QRS_NEXT_CUT()
PTP {E1 28616.934,E2 28616.934}
PTP {X 0,Y 607.906,A -85,B 0,C 180,E1 28616.934,E2 28616.934,E3 0,E4 0,E5 0,E6 0}
QRS_SPEED_INIT()
LIN {X 0,Y 607.906,Z 931,A -85,B 0,C 180,E1 28616.934,E2 28616.934,E3 0,E4 0,E5 0,E6 0} C_VEL
LIN {X 0,Y 607.906,Z 437.153,A -85,B 0,C 180,E1 28616.934,E2 28616.934} C_VEL
LIN {X 0,Y 607.906,Z 429.074,A -85,B 0,C 180,E1 28616.934,E2 28616.934} C_VEL
LIN {X 0,Y 607.894,Z 427.074,A -85,B 0,C 180,E1 28616.745,E2 28616.745} C_VEL
LIN {X 0,Y 607.905,Z 427.069,A -85,B 0,C 180,E1 28613.578,E2 28613.578} C_VEL
LIN {X 0,Y 607.887,Z 427.072,A -85,B 0,C 180,E1 28610.437,E2 28610.437} C_VEL
LIN {X 0,Y 607.904,Z 427.071,A -85,B 0,C 180,E1 28607.364,E2 28607.364} C_VEL
LIN {X 0,Y 607.887,Z 427.071,A -85,B 0,C 180,E1 28604.199,E2 28604.199} C_VEL
LIN {X 0,Y 607.905,Z 427.073,A -85,B 0,C 180,E1 28601.038,E2 28601.038} C_VEL
LIN {X 0,Y 607.891,Z 427.069,A -85,B 0,C 180,E1 28597.873,E2 28597.873} C_VEL
LIN {X 0,Y 607.916,Z 427.076,A -85,B 0,C 180,E1 28594.682,E2 28594.682} C_VEL
LIN {X 0,Y 607.915,Z 427.066,A -85,B 0,C 180,E1 28591.405,E2 28591.405} C_VEL
LIN {X 0,Y 607.89,Z 427.074,A -85,B 0,C 180,E1 28588.13,E2 28588.13} C_VEL
LIN {X 0,Y 607.908,Z 427.069,A -85,B 0,C 180,E1 28584.993,E2 28584.993} C_VEL
LIN {X 0,Y 607.885,Z 427.073,A -85,B 0,C 180,E1 28581.834,E2 28581.834} C_VEL
LIN {X 0,Y 607.906,Z 427.072,A -85,B 0,C 180,E1 28578.734,E2 28578.734} C_VEL
LIN {X 0,Y 607.913,Z 427.228,A -85,B 0,C 180,E1 28576.359,E2 28576.359} C_VEL
LIN {X 0,Y 607.865,Z 452.581,A -85,B 0,C 180,E1 28573.635,E2 28573.635} C_VEL
LIN {X 0,Y 607.881,Z 483.645,A -85,B 0,C 180,E1 28570.395,E2 28570.395} C_VEL
LIN {X 0,Y 607.891,Z 513.28,A -85,B 0,C 180,E1 28567.368,E2 28567.368} C_VEL
LIN {X 0,Y 607.869,Z 545.119,A -85,B 0,C 180,E1 28564.171,E2 28564.171} C_VEL
LIN {X 0,Y 607.907,Z 557.135,A -85,B 0,C 180,E1 28563.013,E2 28563.013} C_VEL
LIN {X 0,Y 607.887,Z 667.971,A -85,B 0,C 180,E1 28561.672,E2 28561.672} C_VEL
LIN {X 0,Y 607.914,Z 683.089,A -85,B 0,C 180,E1 28561.314,E2 28561.314} C_VEL
LIN {X 0,Y 607.919,Z 697.917,A -85,B 0,C 180,E1 28560.764,E2 28560.764} C_VEL
LIN {X 0,Y 607.887,Z 710.969,A -85,B 0,C 180,E1 28560.097,E2 28560.097} C_VEL
LIN {X 0,Y 607.919,Z 723.773,A -85,B 0,C 180,E1 28559.241,E2 28559.241} C_VEL
LIN {X 0,Y 607.918,Z 735.573,A -85,B 0,C 180,E1 28558.22,E2 28558.22} C_VEL
LIN {X 0,Y 607.918,Z 745.62,A -85,B 0,C 180,E1 28557.103,E2 28557.103} C_VEL
LIN {X 0,Y 607.916,Z 753.763,A -85,B 0,C 180,E1 28555.944,E2 28555.944} C_VEL
LIN {X 0,Y 607.918,Z 760.511,A -85,B 0,C 180,E1 28554.693,E2 28554.693} C_VEL
LIN {X 0,Y 607.918,Z 765.691,A -85,B 0,C 180,E1 28553.352,E2 28553.352} C_VEL
LIN {X 0,Y 607.917,Z 769.064,A -85,B 0,C 180,E1 28552.024,E2 28552.024} C_VEL
LIN {X 0,Y 607.917,Z 770.86,A -85,B 0,C 180,E1 28550.507,E2 28550.507} C_VEL
LIN {X 0,Y 607.916,Z 770.652,A -85,B 0,C 180,E1 28549.105,E2 28549.105} C_VEL
LIN {X 0,Y 607.915,Z 768.709,A -85,B 0,C 180,E1 28547.714,E2 28547.714} C_VEL
LIN {X 0,Y 607.919,Z 764.978,A -85,B 0,C 180,E1 28546.335,E2 28546.335} C_VEL
LIN {X 0,Y 607.919,Z 759.759,A -85,B 0,C 180,E1 28545.062,E2 28545.062} C_VEL
LIN {X 0,Y 607.918,Z 752.726,A -85,B 0,C 180,E1 28543.797,E2 28543.797} C_VEL
LIN {X 0,Y 607.919,Z 743.434,A -85,B 0,C 180,E1 28542.539,E2 28542.539} C_VEL
LIN {X 0,Y 607.917,Z 733.34,A -85,B 0,C 180,E1 28541.479,E2 28541.479} C_VEL
LIN {X 0,Y 607.917,Z 722.393,A -85,B 0,C 180,E1 28540.567,E2 28540.567} C_VEL
LIN {X 0,Y 607.901,Z 709.969,A -85,B 0,C 180,E1 28539.753,E2 28539.753} C_VEL
LIN {X 0,Y 607.919,Z 696.486,A -85,B 0,C 180,E1 28539.084,E2 28539.084} C_VEL
LIN {X 0,Y 607.919,Z 682.685,A -85,B 0,C 180,E1 28538.584,E2 28538.584} C_VEL
LIN {X 0,Y 607.915,Z 667.346,A -85,B 0,C 180,E1 28538.227,E2 28538.227} C_VEL
LIN {X 0,Y 607.917,Z 556.808,A -85,B 0,C 180,E1 28536.884,E2 28536.884} C_VEL
LIN {X 0,Y 607.915,Z 525.458,A -85,B 0,C 180,E1 28533.772,E2 28533.772} C_VEL
LIN {X 0,Y 607.88,Z 494.79,A -85,B 0,C 180,E1 28530.66,E2 28530.66} C_VEL
LIN {X 0,Y 607.901,Z 464.7,A -85,B 0,C 180,E1 28527.549,E2 28527.549} C_VEL
LIN {X 0,Y 607.919,Z 435.21,A -85,B 0,C 180,E1 28524.431,E2 28524.431} C_VEL
LIN {X 0,Y 607.9,Z 427.179,A -85,B 0,C 180,E1 28523.531,E2 28523.531} C_VEL
LIN {X 0,Y 607.841,Z 427.076,A -85,B 0,C 180,E1 28520.628,E2 28520.628} C_VEL
LIN {X 0,Y 607.911,Z 427.078,A -85,B 0,C 180,E1 28517.557,E2 28517.557} C_VEL
LIN {X 0,Y 607.836,Z 427.076,A -85,B 0,C 180,E1 28514.545,E2 28514.545} C_VEL
LIN {X 0,Y 607.919,Z 427.077,A -85,B 0,C 180,E1 28511.492,E2 28511.492} C_VEL
LIN {X 0,Y 607.831,Z 427.077,A -85,B 0,C 180,E1 28508.48,E2 28508.48} C_VEL
LIN {X 0,Y 607.906,Z 427.077,A -85,B 0,C 180,E1 28505.444,E2 28505.444} C_VEL
LIN {X 0,Y 607.827,Z 427.077,A -85,B 0,C 180,E1 28502.455,E2 28502.455} C_VEL
LIN {X 0,Y 607.883,Z 427.077,A -85,B 0,C 180,E1 28499.53,E2 28499.53} C_VEL
LIN {X 0,Y 607.829,Z 427.077,A -85,B 0,C 180,E1 28496.447,E2 28496.447} C_VEL
LIN {X 0,Y 607.87,Z 427.077,A -85,B 0,C 180,E1 28493.547,E2 28493.547} C_VEL
LIN {X 0,Y 607.839,Z 427.077,A -85,B 0,C 180,E1 28490.462,E2 28490.462} C_VEL
LIN {X 0,Y 607.846,Z 427.077,A -85,B 0,C 180,E1 28487.718,E2 28487.718} C_VEL
LIN {X 0,Y 607.85,Z 427.076,A -85,B 0,C 180,E1 28484.447,E2 28484.447} C_VEL
LIN {X 0,Y 607.848,Z 427.076,A -85,B 0,C 180,E1 28481.648,E2 28481.648} C_VEL
LIN {X 0,Y 607.853,Z 427.075,A -85,B 0,C 180,E1 28478.314,E2 28478.314} C_VEL
LIN {X 0,Y 607.856,Z 427.076,A -85,B 0,C 180,E1 28475.489,E2 28475.489} C_VEL
LIN {X 0,Y 607.857,Z 427.074,A -85,B 0,C 180,E1 28472.205,E2 28472.205} C_VEL
LIN {X 0,Y 607.864,Z 427.076,A -85,B 0,C 180,E1 28469.333,E2 28469.333} C_VEL
LIN {X 0,Y 607.859,Z 427.073,A -85,B 0,C 180,E1 28466.052,E2 28466.052} C_VEL
LIN {X 0,Y 607.875,Z 427.076,A -85,B 0,C 180,E1 28463.149,E2 28463.149} C_VEL
LIN {X 0,Y 607.86,Z 427.073,A -85,B 0,C 180,E1 28459.907,E2 28459.907} C_VEL
LIN {X 0,Y 607.891,Z 427.076,A -85,B 0,C 180,E1 28456.926,E2 28456.926} C_VEL
LIN {X 0,Y 607.86,Z 427.073,A -85,B 0,C 180,E1 28453.702,E2 28453.702} C_VEL
LIN {X 0,Y 607.908,Z 427.077,A -85,B 0,C 180,E1 28450.711,E2 28450.711} C_VEL
LIN {X 0,Y 607.863,Z 427.072,A -85,B 0,C 180,E1 28447.562,E2 28447.562} C_VEL
LIN {X 0,Y 607.911,Z 427.078,A -85,B 0,C 180,E1 28444.528,E2 28444.528} C_VEL
LIN {X 0,Y 607.866,Z 427.072,A -85,B 0,C 180,E1 28441.414,E2 28441.414} C_VEL
LIN {X 0,Y 607.915,Z 427.075,A -85,B 0,C 180,E1 28438.304,E2 28438.304} C_VEL
LIN {X 0,Y 607.867,Z 427.073,A -85,B 0,C 180,E1 28435.188,E2 28435.188} C_VEL
LIN {X 0,Y 607.913,Z 427.072,A -85,B 0,C 180,E1 28432.059,E2 28432.059} C_VEL
LIN {X 0,Y 607.87,Z 427.073,A -85,B 0,C 180,E1 28429,E2 28429} C_VEL
LIN {X 0,Y 607.912,Z 427.071,A -85,B 0,C 180,E1 28425.912,E2 28425.912} C_VEL
LIN {X 0,Y 607.875,Z 427.073,A -85,B 0,C 180,E1 28422.874,E2 28422.874} C_VEL
LIN {X 0,Y 607.912,Z 427.069,A -85,B 0,C 180,E1 28419.694,E2 28419.694} C_VEL
LIN {X 0,Y 607.885,Z 427.074,A -85,B 0,C 180,E1 28416.544,E2 28416.544} C_VEL
LIN {X 0,Y 607.904,Z 427.067,A -85,B 0,C 180,E1 28413.267,E2 28413.267} C_VEL
LIN {X 0,Y 607.915,Z 427.076,A -85,B 0,C 180,E1 28410,E2 28410} C_VEL
LIN {X 0,Y 607.885,Z 427.07,A -85,B 0,C 180,E1 28406.789,E2 28406.789} C_VEL
LIN {X 0,Y 607.906,Z 427.073,A -85,B 0,C 180,E1 28403.693,E2 28403.693} C_VEL
LIN {X 0,Y 607.886,Z 427.071,A -85,B 0,C 180,E1 28400.588,E2 28400.588} C_VEL
LIN {X 0,Y 607.903,Z 427.072,A -85,B 0,C 180,E1 28397.465,E2 28397.465} C_VEL
LIN {X 0,Y 607.889,Z 427.073,A -85,B 0,C 180,E1 28394.317,E2 28394.317} C_VEL
LIN {X 0,Y 607.906,Z 427.069,A -85,B 0,C 180,E1 28391.123,E2 28391.123} C_VEL
LIN {X 0,Y 607.902,Z 427.075,A -85,B 0,C 180,E1 28387.963,E2 28387.963} C_VEL
LIN {X 0,Y 607.909,Z 427.067,A -85,B 0,C 180,E1 28384.677,E2 28384.677} C_VEL
LIN {X 0,Y 607.902,Z 427.076,A -85,B 0,C 180,E1 28381.426,E2 28381.426} C_VEL
LIN {X 0,Y 607.906,Z 427.311,A -85,B 0,C 180,E1 28379.783,E2 28379.783} C_VEL
LIN {X 0,Y 607.918,Z 435.341,A -85,B 0,C 180,E1 28379.195,E2 28379.195} C_VEL
LIN {X 0,Y 607.898,Z 480.356,A -85,B 0,C 180,E1 28376.155,E2 28376.155} C_VEL
LIN {X 0,Y 607.881,Z 526.04,A -85,B 0,C 180,E1 28373.149,E2 28373.149} C_VEL
LIN {X 0,Y 607.914,Z 539.004,A -85,B 0,C 180,E1 28372.33,E2 28372.33} C_VEL
LIN {X 0,Y 607.912,Z 748.311,A -85,B 0,C 180,E1 28369.705,E2 28369.705} C_VEL
LIN {X 0,Y 607.888,Z 766.586,A -85,B 0,C 180,E1 28369.306,E2 28369.306} C_VEL
LIN {X 0,Y 607.901,Z 784.762,A -85,B 0,C 180,E1 28368.732,E2 28368.732} C_VEL
LIN {X 0,Y 607.893,Z 803.057,A -85,B 0,C 180,E1 28367.963,E2 28367.963} C_VEL
LIN {X 0,Y 607.919,Z 819.788,A -85,B 0,C 180,E1 28367.073,E2 28367.073} C_VEL
LIN {X 0,Y 607.916,Z 835.64,A -85,B 0,C 180,E1 28366.041,E2 28366.041} C_VEL
LIN {X 0,Y 607.917,Z 850.561,A -85,B 0,C 180,E1 28364.867,E2 28364.867} C_VEL
LIN {X 0,Y 607.918,Z 864.218,A -85,B 0,C 180,E1 28363.582,E2 28363.582} C_VEL
LIN {X 0,Y 607.918,Z 876.905,A -85,B 0,C 180,E1 28362.153,E2 28362.153} C_VEL
LIN {X 0,Y 607.911,Z 888.224,A -85,B 0,C 180,E1 28360.615,E2 28360.615} C_VEL
LIN {X 0,Y 607.918,Z 897.988,A -85,B 0,C 180,E1 28358.989,E2 28358.989} C_VEL
LIN {X 0,Y 607.909,Z 905.863,A -85,B 0,C 180,E1 28357.35,E2 28357.35} C_VEL
LIN {X 0,Y 607.906,Z 912.107,A -85,B 0,C 180,E1 28355.664,E2 28355.664} C_VEL
LIN {X 0,Y 607.917,Z 916.872,A -85,B 0,C 180,E1 28353.867,E2 28353.867} C_VEL
LIN {X 0,Y 607.916,Z 919.787,A -85,B 0,C 180,E1 28352.074,E2 28352.074} C_VEL
LIN {X 0,Y 607.907,Z 920.94,A -85,B 0,C 180,E1 28350.283,E2 28350.283} C_VEL
LIN {X 0,Y 607.915,Z 920.348,A -85,B 0,C 180,E1 28348.492,E2 28348.492} C_VEL
LIN {X 0,Y 607.908,Z 918.005,A -85,B 0,C 180,E1 28346.7,E2 28346.7} C_VEL
LIN {X 0,Y 607.905,Z 914.096,A -85,B 0,C 180,E1 28344.999,E2 28344.999} C_VEL
LIN {X 0,Y 607.912,Z 908.468,A -85,B 0,C 180,E1 28343.294,E2 28343.294} C_VEL
LIN {X 0,Y 607.915,Z 901.423,A -85,B 0,C 180,E1 28341.678,E2 28341.678} C_VEL
LIN {X 0,Y 607.911,Z 892.509,A -85,B 0,C 180,E1 28340.055,E2 28340.055} C_VEL
LIN {X 0,Y 607.919,Z 882.145,A -85,B 0,C 180,E1 28338.521,E2 28338.521} C_VEL
LIN {X 0,Y 607.914,Z 870.346,A -85,B 0,C 180,E1 28337.075,E2 28337.075} C_VEL
LIN {X 0,Y 607.917,Z 857.089,A -85,B 0,C 180,E1 28335.717,E2 28335.717} C_VEL
LIN {X 0,Y 607.917,Z 842.235,A -85,B 0,C 180,E1 28334.449,E2 28334.449} C_VEL
LIN {X 0,Y 607.917,Z 826.219,A -85,B 0,C 180,E1 28333.321,E2 28333.321} C_VEL
LIN {X 0,Y 607.898,Z 810.027,A -85,B 0,C 180,E1 28332.384,E2 28332.384} C_VEL
LIN {X 0,Y 607.913,Z 793.065,A -85,B 0,C 180,E1 28331.592,E2 28331.592} C_VEL
LIN {X 0,Y 607.886,Z 775.227,A -85,B 0,C 180,E1 28330.944,E2 28330.944} C_VEL
LIN {X 0,Y 607.899,Z 756.387,A -85,B 0,C 180,E1 28330.45,E2 28330.45} C_VEL
LIN {X 0,Y 607.919,Z 736.792,A -85,B 0,C 180,E1 28330.128,E2 28330.128} C_VEL
LIN {X 0,Y 607.915,Z 538.331,A -85,B 0,C 180,E1 28327.645,E2 28327.645} C_VEL
LIN {X 0,Y 607.904,Z 491.389,A -85,B 0,C 180,E1 28324.578,E2 28324.578} C_VEL
LIN {X 0,Y 607.919,Z 444.131,A -85,B 0,C 180,E1 28321.405,E2 28321.405} C_VEL
LIN {X 0,Y 607.907,Z 427.395,A -85,B 0,C 180,E1 28320.232,E2 28320.232} C_VEL
LIN {X 0,Y 607.912,Z 427.067,A -85,B 0,C 180,E1 28319.339,E2 28319.339} C_VEL
LIN {X 0,Y 607.906,Z 427.076,A -85,B 0,C 180,E1 28316.112,E2 28316.112} C_VEL
LIN {X 0,Y 607.902,Z 427.069,A -85,B 0,C 180,E1 28312.912,E2 28312.912} C_VEL
LIN {X 0,Y 607.895,Z 427.073,A -85,B 0,C 180,E1 28309.729,E2 28309.729} C_VEL
LIN {X 0,Y 607.898,Z 427.071,A -85,B 0,C 180,E1 28306.566,E2 28306.566} C_VEL
LIN {X 0,Y 607.893,Z 427.071,A -85,B 0,C 180,E1 28303.434,E2 28303.434} C_VEL
LIN {X 0,Y 607.901,Z 427.073,A -85,B 0,C 180,E1 28300.27,E2 28300.27} C_VEL
LIN {X 0,Y 607.899,Z 427.068,A -85,B 0,C 180,E1 28297.088,E2 28297.088} C_VEL
LIN {X 0,Y 607.913,Z 427.078,A -85,B 0,C 180,E1 28293.84,E2 28293.84} C_VEL
LIN {X 0,Y 607.908,Z 427.067,A -85,B 0,C 180,E1 28290.546,E2 28290.546} C_VEL
LIN {X 0,Y 607.894,Z 427.073,A -85,B 0,C 180,E1 28287.316,E2 28287.316} C_VEL
LIN {X 0,Y 607.901,Z 427.07,A -85,B 0,C 180,E1 28284.176,E2 28284.176} C_VEL
LIN {X 0,Y 607.891,Z 427.071,A -85,B 0,C 180,E1 28281.012,E2 28281.012} C_VEL
LIN {X 0,Y 607.901,Z 427.072,A -85,B 0,C 180,E1 28277.913,E2 28277.913} C_VEL
LIN {X 0,Y 607.89,Z 427.071,A -85,B 0,C 180,E1 28274.868,E2 28274.868} C_VEL
LIN {X 0,Y 607.9,Z 427.072,A -85,B 0,C 180,E1 28271.768,E2 28271.768} C_VEL
LIN {X 0,Y 607.89,Z 427.071,A -85,B 0,C 180,E1 28268.688,E2 28268.688} C_VEL
LIN {X 0,Y 607.903,Z 427.073,A -85,B 0,C 180,E1 28265.569,E2 28265.569} C_VEL
LIN {X 0,Y 607.892,Z 427.07,A -85,B 0,C 180,E1 28262.451,E2 28262.451} C_VEL
LIN {X 0,Y 607.91,Z 427.076,A -85,B 0,C 180,E1 28259.246,E2 28259.246} C_VEL
LIN {X 0,Y 607.894,Z 427.074,A -85,B 0,C 180,E1 28256.745,E2 28256.745} C_VEL
LIN {X 0,Y 606.888,Z 427.198,A -85,B 0,C 180,E1 28256.019,E2 28256.019} C_VEL
LIN {X 0,Y 600.49,Z 427.993,A -85,B 0,C 180,E1 28253.983,E2 28253.983} C_VEL
LIN {X 0,Y 599.964,Z 428.06,A -85,B 0,C 180,E1 28253.453,E2 28253.453} C_VEL
LIN {X 0,Y 599.949,Z 428.059,A -85,B 0,C 180,E1 28250.309,E2 28250.309} C_VEL
LIN {X 0,Y 599.968,Z 428.063,A -85,B 0,C 180,E1 28247.096,E2 28247.096} C_VEL
LIN {X 0,Y 599.962,Z 428.057,A -85,B 0,C 180,E1 28243.84,E2 28243.84} C_VEL
LIN {X 0,Y 599.961,Z 428.064,A -85,B 0,C 180,E1 28240.53,E2 28240.53} C_VEL
LIN {X 0,Y 599.973,Z 428.057,A -85,B 0,C 180,E1 28237.358,E2 28237.358} C_VEL
LIN {X 0,Y 599.948,Z 428.062,A -85,B 0,C 180,E1 28234.151,E2 28234.151} C_VEL
LIN {X 0,Y 599.966,Z 428.06,A -85,B 0,C 180,E1 28230.99,E2 28230.99} C_VEL
LIN {X 0,Y 599.946,Z 428.06,A -85,B 0,C 180,E1 28227.846,E2 28227.846} C_VEL
LIN {X 0,Y 599.969,Z 428.063,A -85,B 0,C 180,E1 28224.67,E2 28224.67} C_VEL
LIN {X 0,Y 599.949,Z 428.06,A -85,B 0,C 180,E1 28221.563,E2 28221.563} C_VEL
LIN {X 0,Y 599.977,Z 428.065,A -85,B 0,C 180,E1 28218.296,E2 28218.296} C_VEL
LIN {X 0,Y 600.001,Z 428.308,A -85,B 0,C 180,E1 28216.611,E2 28216.611} C_VEL
LIN {X 0,Y 600.305,Z 432.323,A -85,B 0,C 180,E1 28216.141,E2 28216.141} C_VEL
LIN {X 0,Y 600.213,Z 462.032,A -85,B 0,C 180,E1 28212.947,E2 28212.947} C_VEL
LIN {X 0,Y 600.131,Z 492.243,A -85,B 0,C 180,E1 28209.774,E2 28209.774} C_VEL
LIN {X 0,Y 600.074,Z 523.353,A -85,B 0,C 180,E1 28206.57,E2 28206.57} C_VEL
LIN {X 0,Y 599.98,Z 553.885,A -85,B 0,C 180,E1 28203.477,E2 28203.477} C_VEL
LIN {X 0,Y 600.063,Z 557.379,A -85,B 0,C 180,E1 28203.181,E2 28203.181} C_VEL
LIN {X 0,Y 600.05,Z 668.429,A -85,B 0,C 180,E1 28201.819,E2 28201.819} C_VEL
LIN {X 0,Y 600.059,Z 683.234,A -85,B 0,C 180,E1 28201.461,E2 28201.461} C_VEL
LIN {X 0,Y 600.039,Z 698.352,A -85,B 0,C 180,E1 28200.889,E2 28200.889} C_VEL
LIN {X 0,Y 599.979,Z 711.224,A -85,B 0,C 180,E1 28200.217,E2 28200.217} C_VEL
LIN {X 0,Y 599.985,Z 723.853,A -85,B 0,C 180,E1 28199.358,E2 28199.358} C_VEL
LIN {X 0,Y 599.959,Z 735.895,A -85,B 0,C 180,E1 28198.298,E2 28198.298} C_VEL
LIN {X 0,Y 599.941,Z 746.161,A -85,B 0,C 180,E1 28197.131,E2 28197.131} C_VEL
LIN {X 0,Y 599.927,Z 754.564,A -85,B 0,C 180,E1 28195.891,E2 28195.891} C_VEL
LIN {X 0,Y 599.921,Z 761.097,A -85,B 0,C 180,E1 28194.624,E2 28194.624} C_VEL
LIN {X 0,Y 599.915,Z 766.428,A -85,B 0,C 180,E1 28193.162,E2 28193.162} C_VEL
LIN {X 0,Y 599.916,Z 769.618,A -85,B 0,C 180,E1 28191.715,E2 28191.715} C_VEL
LIN {X 0,Y 599.919,Z 770.906,A -85,B 0,C 180,E1 28190.385,E2 28190.385} C_VEL
LIN {X 0,Y 599.914,Z 770.563,A -85,B 0,C 180,E1 28188.965,E2 28188.965} C_VEL
LIN {X 0,Y 599.915,Z 768.439,A -85,B 0,C 180,E1 28187.558,E2 28187.558} C_VEL
LIN {X 0,Y 599.919,Z 764.544,A -85,B 0,C 180,E1 28186.16,E2 28186.16} C_VEL
LIN {X 0,Y 599.921,Z 758.689,A -85,B 0,C 180,E1 28184.773,E2 28184.773} C_VEL
LIN {X 0,Y 599.932,Z 751.258,A -85,B 0,C 180,E1 28183.493,E2 28183.493} C_VEL
LIN {X 0,Y 599.948,Z 742.392,A -85,B 0,C 180,E1 28182.317,E2 28182.317} C_VEL
LIN {X 0,Y 599.969,Z 731.526,A -85,B 0,C 180,E1 28181.195,E2 28181.195} C_VEL
LIN {X 0,Y 599.992,Z 719.4,A -85,B 0,C 180,E1 28180.223,E2 28180.223} C_VEL
LIN {X 0,Y 600.009,Z 706.382,A -85,B 0,C 180,E1 28179.419,E2 28179.419} C_VEL
LIN {X 0,Y 600.047,Z 693.632,A -85,B 0,C 180,E1 28178.818,E2 28178.818} C_VEL
LIN {X 0,Y 600.068,Z 678.136,A -85,B 0,C 180,E1 28178.305,E2 28178.305} C_VEL
LIN {X 0,Y 600.083,Z 663.073,A -85,B 0,C 180,E1 28178.006,E2 28178.006} C_VEL
LIN {X 0,Y 600.032,Z 556.838,A -85,B 0,C 180,E1 28176.712,E2 28176.712} C_VEL
LIN {X 0,Y 600.07,Z 525.261,A -85,B 0,C 180,E1 28173.534,E2 28173.534} C_VEL
LIN {X 0,Y 600.129,Z 493.692,A -85,B 0,C 180,E1 28170.286,E2 28170.286} C_VEL
LIN {X 0,Y 600.201,Z 463.661,A -85,B 0,C 180,E1 28167.135,E2 28167.135} C_VEL
LIN {X 0,Y 600.301,Z 434.227,A -85,B 0,C 180,E1 28163.977,E2 28163.977} C_VEL
LIN {X 0,Y 600.118,Z 429.008,A -85,B 0,C 180,E1 28163.398,E2 28163.398} C_VEL
LIN {X 0,Y 599.928,Z 428.099,A -85,B 0,C 180,E1 28163.204,E2 28163.204} C_VEL
LIN {X 0,Y 599.916,Z 428.065,A -85,B 0,C 180,E1 28160.309,E2 28160.309} C_VEL
LIN {X 0,Y 599.912,Z 428.066,A -85,B 0,C 180,E1 28156.997,E2 28156.997} C_VEL
LIN {X 0,Y 599.916,Z 428.065,A -85,B 0,C 180,E1 28154.137,E2 28154.137} C_VEL
LIN {X 0,Y 599.903,Z 428.066,A -85,B 0,C 180,E1 28150.832,E2 28150.832} C_VEL
LIN {X 0,Y 599.907,Z 428.065,A -85,B 0,C 180,E1 28148.078,E2 28148.078} C_VEL
LIN {X 0,Y 599.901,Z 428.066,A -85,B 0,C 180,E1 28144.743,E2 28144.743} C_VEL
LIN {X 0,Y 599.903,Z 428.066,A -85,B 0,C 180,E1 28141.965,E2 28141.965} C_VEL
LIN {X 0,Y 599.898,Z 428.066,A -85,B 0,C 180,E1 28138.667,E2 28138.667} C_VEL
LIN {X 0,Y 599.897,Z 428.066,A -85,B 0,C 180,E1 28135.931,E2 28135.931} C_VEL
LIN {X 0,Y 599.909,Z 428.065,A -85,B 0,C 180,E1 28132.65,E2 28132.65} C_VEL
LIN {X 0,Y 599.901,Z 428.066,A -85,B 0,C 180,E1 28129.833,E2 28129.833} C_VEL
LIN {X 0,Y 599.92,Z 428.065,A -85,B 0,C 180,E1 28126.608,E2 28126.608} C_VEL
LIN {X 0,Y 599.904,Z 428.065,A -85,B 0,C 180,E1 28123.764,E2 28123.764} C_VEL
LIN {X 0,Y 599.929,Z 428.063,A -85,B 0,C 180,E1 28120.537,E2 28120.537} C_VEL
LIN {X 0,Y 599.908,Z 428.065,A -85,B 0,C 180,E1 28117.657,E2 28117.657} C_VEL
LIN {X 0,Y 599.931,Z 428.061,A -85,B 0,C 180,E1 28114.402,E2 28114.402} C_VEL
LIN {X 0,Y 599.911,Z 428.065,A -85,B 0,C 180,E1 28111.557,E2 28111.557} C_VEL
LIN {X 0,Y 599.942,Z 428.061,A -85,B 0,C 180,E1 28108.358,E2 28108.358} C_VEL
LIN {X 0,Y 599.918,Z 428.063,A -85,B 0,C 180,E1 28105.4,E2 28105.4} C_VEL
LIN {X 0,Y 599.93,Z 428.062,A -85,B 0,C 180,E1 28102.082,E2 28102.082} C_VEL
LIN {X 0,Y 599.937,Z 428.064,A -85,B 0,C 180,E1 28099.096,E2 28099.096} C_VEL
LIN {X 0,Y 599.926,Z 428.061,A -85,B 0,C 180,E1 28095.863,E2 28095.863} C_VEL
LIN {X 0,Y 599.96,Z 428.066,A -85,B 0,C 180,E1 28092.806,E2 28092.806} C_VEL
LIN {X 0,Y 599.924,Z 428.06,A -85,B 0,C 180,E1 28089.594,E2 28089.594} C_VEL
LIN {X 0,Y 599.976,Z 428.065,A -85,B 0,C 180,E1 28086.507,E2 28086.507} C_VEL
LIN {X 0,Y 599.925,Z 428.062,A -85,B 0,C 180,E1 28083.32,E2 28083.32} C_VEL
LIN {X 0,Y 599.975,Z 428.06,A -85,B 0,C 180,E1 28080.191,E2 28080.191} C_VEL
LIN {X 0,Y 599.928,Z 428.062,A -85,B 0,C 180,E1 28077.134,E2 28077.134} C_VEL
LIN {X 0,Y 599.977,Z 428.058,A -85,B 0,C 180,E1 28073.974,E2 28073.974} C_VEL
LIN {X 0,Y 599.934,Z 428.062,A -85,B 0,C 180,E1 28070.89,E2 28070.89} C_VEL
LIN {X 0,Y 599.975,Z 428.057,A -85,B 0,C 180,E1 28067.684,E2 28067.684} C_VEL
LIN {X 0,Y 599.961,Z 428.064,A -85,B 0,C 180,E1 28064.421,E2 28064.421} C_VEL
LIN {X 0,Y 599.942,Z 428.06,A -85,B 0,C 180,E1 28061.136,E2 28061.136} C_VEL
LIN {X 0,Y 599.972,Z 428.063,A -85,B 0,C 180,E1 28057.978,E2 28057.978} C_VEL
LIN {X 0,Y 599.941,Z 428.061,A -85,B 0,C 180,E1 28054.819,E2 28054.819} C_VEL
LIN {X 0,Y 599.97,Z 428.06,A -85,B 0,C 180,E1 28051.644,E2 28051.644} C_VEL
LIN {X 0,Y 599.945,Z 428.061,A -85,B 0,C 180,E1 28048.558,E2 28048.558} C_VEL
LIN {X 0,Y 599.971,Z 428.057,A -85,B 0,C 180,E1 28045.37,E2 28045.37} C_VEL
LIN {X 0,Y 599.96,Z 428.064,A -85,B 0,C 180,E1 28042.173,E2 28042.173} C_VEL
LIN {X 0,Y 599.959,Z 428.058,A -85,B 0,C 180,E1 28038.831,E2 28038.831} C_VEL
LIN {X 0,Y 599.968,Z 428.063,A -85,B 0,C 180,E1 28035.638,E2 28035.638} C_VEL
LIN {X 0,Y 599.951,Z 428.061,A -85,B 0,C 180,E1 28032.414,E2 28032.414} C_VEL
LIN {X 0,Y 599.962,Z 428.061,A -85,B 0,C 180,E1 28029.293,E2 28029.293} C_VEL
LIN {X 0,Y 599.954,Z 428.063,A -85,B 0,C 180,E1 28026.155,E2 28026.155} C_VEL
LIN {X 0,Y 599.968,Z 428.056,A -85,B 0,C 180,E1 28022.908,E2 28022.908} C_VEL
LIN {X 0,Y 599.982,Z 428.256,A -85,B 0,C 180,E1 28020.157,E2 28020.157} C_VEL
LIN {X 0,Y 600.653,Z 431.523,A -85,B 0,C 180,E1 28019.85,E2 28019.85} C_VEL
LIN {X 0,Y 600.505,Z 477.206,A -85,B 0,C 180,E1 28016.716,E2 28016.716} C_VEL
LIN {X 0,Y 600.351,Z 524.464,A -85,B 0,C 180,E1 28013.56,E2 28013.56} C_VEL
LIN {X 0,Y 600.433,Z 539.199,A -85,B 0,C 180,E1 28012.62,E2 28012.62} C_VEL
LIN {X 0,Y 600.372,Z 748.311,A -85,B 0,C 180,E1 28009.963,E2 28009.963} C_VEL
LIN {X 0,Y 600.309,Z 767.215,A -85,B 0,C 180,E1 28009.541,E2 28009.541} C_VEL
LIN {X 0,Y 600.273,Z 785.404,A -85,B 0,C 180,E1 28008.954,E2 28008.954} C_VEL
LIN {X 0,Y 600.211,Z 803.054,A -85,B 0,C 180,E1 28008.201,E2 28008.201} C_VEL
LIN {X 0,Y 600.18,Z 819.704,A -85,B 0,C 180,E1 28007.305,E2 28007.305} C_VEL
LIN {X 0,Y 600.122,Z 835.639,A -85,B 0,C 180,E1 28006.255,E2 28006.255} C_VEL
LIN {X 0,Y 600.069,Z 850.562,A -85,B 0,C 180,E1 28005.066,E2 28005.066} C_VEL
LIN {X 0,Y 600.02,Z 864.018,A -85,B 0,C 180,E1 28003.786,E2 28003.786} C_VEL
LIN {X 0,Y 599.985,Z 876.906,A -85,B 0,C 180,E1 28002.316,E2 28002.316} C_VEL
LIN {X 0,Y 599.953,Z 888.224,A -85,B 0,C 180,E1 28000.758,E2 28000.758} C_VEL
LIN {X 0,Y 599.935,Z 897.989,A -85,B 0,C 180,E1 27999.11,E2 27999.11} C_VEL
LIN {X 0,Y 599.92,Z 906.042,A -85,B 0,C 180,E1 27997.406,E2 27997.406} C_VEL
LIN {X 0,Y 599.91,Z 912.409,A -85,B 0,C 180,E1 27995.643,E2 27995.643} C_VEL
LIN {X 0,Y 599.918,Z 916.873,A -85,B 0,C 180,E1 27993.918,E2 27993.918} C_VEL
LIN {X 0,Y 599.917,Z 919.787,A -85,B 0,C 180,E1 27992.101,E2 27992.101} C_VEL
LIN {X 0,Y 599.907,Z 920.94,A -85,B 0,C 180,E1 27990.287,E2 27990.287} C_VEL
LIN {X 0,Y 599.915,Z 920.348,A -85,B 0,C 180,E1 27988.472,E2 27988.472} C_VEL
LIN {X 0,Y 599.907,Z 918.006,A -85,B 0,C 180,E1 27986.656,E2 27986.656} C_VEL
LIN {X 0,Y 599.908,Z 914.097,A -85,B 0,C 180,E1 27984.932,E2 27984.932} C_VEL
LIN {X 0,Y 599.919,Z 908.468,A -85,B 0,C 180,E1 27983.204,E2 27983.204} C_VEL
LIN {X 0,Y 599.927,Z 901.424,A -85,B 0,C 180,E1 27981.567,E2 27981.567} C_VEL
LIN {X 0,Y 599.942,Z 892.51,A -85,B 0,C 180,E1 27979.922,E2 27979.922} C_VEL
LIN {X 0,Y 599.969,Z 882.146,A -85,B 0,C 180,E1 27978.367,E2 27978.367} C_VEL
LIN {X 0,Y 600,Z 870.347,A -85,B 0,C 180,E1 27976.901,E2 27976.901} C_VEL
LIN {X 0,Y 600.049,Z 856.752,A -85,B 0,C 180,E1 27975.493,E2 27975.493} C_VEL
LIN {X 0,Y 600.103,Z 842.234,A -85,B 0,C 180,E1 27974.242,E2 27974.242} C_VEL
LIN {X 0,Y 600.164,Z 826.222,A -85,B 0,C 180,E1 27973.1,E2 27973.1} C_VEL
LIN {X 0,Y 600.199,Z 809.035,A -85,B 0,C 180,E1 27972.1,E2 27972.1} C_VEL
LIN {X 0,Y 600.279,Z 791.772,A -85,B 0,C 180,E1 27971.298,E2 27971.298} C_VEL
LIN {X 0,Y 600.297,Z 773.83,A -85,B 0,C 180,E1 27970.652,E2 27970.652} C_VEL
LIN {X 0,Y 600.353,Z 755.31,A -85,B 0,C 180,E1 27970.173,E2 27970.173} C_VEL
LIN {X 0,Y 600.395,Z 735.522,A -85,B 0,C 180,E1 27969.853,E2 27969.853} C_VEL
LIN {X 0,Y 600.381,Z 538.736,A -85,B 0,C 180,E1 27967.368,E2 27967.368} C_VEL
LIN {X 0,Y 600.472,Z 490.601,A -85,B 0,C 180,E1 27964.188,E2 27964.188} C_VEL
LIN {X 0,Y 600.612,Z 444.131,A -85,B 0,C 180,E1 27961.025,E2 27961.025} C_VEL
LIN {X 0,Y 600.43,Z 429.953,A -85,B 0,C 180,E1 27960.029,E2 27960.029} C_VEL
LIN {X 0,Y 599.968,Z 428.159,A -85,B 0,C 180,E1 27959.813,E2 27959.813} C_VEL
LIN {X 0,Y 599.96,Z 428.063,A -85,B 0,C 180,E1 27956.636,E2 27956.636} C_VEL
LIN {X 0,Y 599.963,Z 428.058,A -85,B 0,C 180,E1 27953.443,E2 27953.443} C_VEL
LIN {X 0,Y 599.974,Z 428.066,A -85,B 0,C 180,E1 27950.198,E2 27950.198} C_VEL
LIN {X 0,Y 599.969,Z 428.056,A -85,B 0,C 180,E1 27946.881,E2 27946.881} C_VEL
LIN {X 0,Y 599.958,Z 428.063,A -85,B 0,C 180,E1 27943.674,E2 27943.674} C_VEL
LIN {X 0,Y 599.961,Z 428.059,A -85,B 0,C 180,E1 27940.538,E2 27940.538} C_VEL
LIN {X 0,Y 599.955,Z 428.06,A -85,B 0,C 180,E1 27937.346,E2 27937.346} C_VEL
LIN {X 0,Y 599.963,Z 428.062,A -85,B 0,C 180,E1 27934.168,E2 27934.168} C_VEL
LIN {X 0,Y 599.958,Z 428.058,A -85,B 0,C 180,E1 27930.995,E2 27930.995} C_VEL
LIN {X 0,Y 599.973,Z 428.066,A -85,B 0,C 180,E1 27927.707,E2 27927.707} C_VEL
LIN {X 0,Y 599.971,Z 428.056,A -85,B 0,C 180,E1 27924.412,E2 27924.412} C_VEL
LIN {X 0,Y 599.955,Z 428.062,A -85,B 0,C 180,E1 27921.201,E2 27921.201} C_VEL
LIN {X 0,Y 599.963,Z 428.059,A -85,B 0,C 180,E1 27918.058,E2 27918.058} C_VEL
LIN {X 0,Y 599.952,Z 428.06,A -85,B 0,C 180,E1 27914.97,E2 27914.97} C_VEL
LIN {X 0,Y 599.962,Z 428.061,A -85,B 0,C 180,E1 27911.828,E2 27911.828} C_VEL
LIN {X 0,Y 599.951,Z 428.06,A -85,B 0,C 180,E1 27908.723,E2 27908.723} C_VEL
LIN {X 0,Y 599.965,Z 428.062,A -85,B 0,C 180,E1 27905.547,E2 27905.547} C_VEL
LIN {X 0,Y 599.955,Z 428.058,A -85,B 0,C 180,E1 27902.388,E2 27902.388} C_VEL
LIN {X 0,Y 599.973,Z 428.066,A -85,B 0,C 180,E1 27899.14,E2 27899.14} C_VEL
LIN {X 0,Y 599.971,Z 428.056,A -85,B 0,C 180,E1 27895.795,E2 27895.795} C_VEL
LIN {X 0,Y 599.964,Z 428.06,A -85,B 0,C 180,E1 27893.453,E2 27893.453} C_VEL
LIN {X 0,Y 598.972,Z 428.19,A -85,B 0,C 180,E1 27892.717,E2 27892.717} C_VEL
LIN {X 0,Y 592.53,Z 428.989,A -85,B 0,C 180,E1 27890.653,E2 27890.653} C_VEL
LIN {X 0,Y 592.015,Z 429.046,A -85,B 0,C 180,E1 27890.116,E2 27890.116} C_VEL
LIN {X 0,Y 592.035,Z 429.053,A -85,B 0,C 180,E1 27886.821,E2 27886.821} C_VEL
LIN {X 0,Y 592.034,Z 429.046,A -85,B 0,C 180,E1 27883.517,E2 27883.517} C_VEL
LIN {X 0,Y 592.01,Z 429.051,A -85,B 0,C 180,E1 27880.258,E2 27880.258} C_VEL
LIN {X 0,Y 592.027,Z 429.049,A -85,B 0,C 180,E1 27877.142,E2 27877.142} C_VEL
LIN {X 0,Y 592.008,Z 429.049,A -85,B 0,C 180,E1 27873.952,E2 27873.952} C_VEL
LIN {X 0,Y 592.03,Z 429.052,A -85,B 0,C 180,E1 27870.785,E2 27870.785} C_VEL
LIN {X 0,Y 592.015,Z 429.047,A -85,B 0,C 180,E1 27867.613,E2 27867.613} C_VEL
LIN {X 0,Y 592.032,Z 429.055,A -85,B 0,C 180,E1 27864.325,E2 27864.325} C_VEL
LIN {X 0,Y 592.034,Z 429.047,A -85,B 0,C 180,E1 27861.078,E2 27861.078} C_VEL
LIN {X 0,Y 592.01,Z 429.054,A -85,B 0,C 180,E1 27857.854,E2 27857.854} C_VEL
LIN {X 0,Y 592.075,Z 429.342,A -85,B 0,C 180,E1 27856.882,E2 27856.882} C_VEL
LIN {X 0,Y 592.706,Z 432.831,A -85,B 0,C 180,E1 27856.446,E2 27856.446} C_VEL
LIN {X 0,Y 592.526,Z 462.63,A -85,B 0,C 180,E1 27853.199,E2 27853.199} C_VEL
LIN {X 0,Y 592.359,Z 492.911,A -85,B 0,C 180,E1 27849.975,E2 27849.975} C_VEL
LIN {X 0,Y 592.238,Z 524.271,A -85,B 0,C 180,E1 27846.702,E2 27846.702} C_VEL
LIN {X 0,Y 592.09,Z 555.284,A -85,B 0,C 180,E1 27843.518,E2 27843.518} C_VEL
LIN {X 0,Y 592.194,Z 557.533,A -85,B 0,C 180,E1 27843.357,E2 27843.357} C_VEL
LIN {X 0,Y 592.217,Z 668.509,A -85,B 0,C 180,E1 27841.977,E2 27841.977} C_VEL
LIN {X 0,Y 592.21,Z 682.541,A -85,B 0,C 180,E1 27841.636,E2 27841.636} C_VEL
LIN {X 0,Y 592.166,Z 696.696,A -85,B 0,C 180,E1 27841.109,E2 27841.109} C_VEL
LIN {X 0,Y 592.087,Z 709.865,A -85,B 0,C 180,E1 27840.438,E2 27840.438} C_VEL
LIN {X 0,Y 592.052,Z 723.076,A -85,B 0,C 180,E1 27839.546,E2 27839.546} C_VEL
LIN {X 0,Y 592.007,Z 734.994,A -85,B 0,C 180,E1 27838.5,E2 27838.5} C_VEL
LIN {X 0,Y 591.967,Z 744.768,A -85,B 0,C 180,E1 27837.404,E2 27837.404} C_VEL
LIN {X 0,Y 591.945,Z 752.951,A -85,B 0,C 180,E1 27836.244,E2 27836.244} C_VEL
LIN {X 0,Y 591.927,Z 760.27,A -85,B 0,C 180,E1 27834.872,E2 27834.872} C_VEL
LIN {X 0,Y 591.919,Z 765.538,A -85,B 0,C 180,E1 27833.493,E2 27833.493} C_VEL
LIN {X 0,Y 591.919,Z 768.975,A -85,B 0,C 180,E1 27832.129,E2 27832.129} C_VEL
LIN {X 0,Y 591.916,Z 770.781,A -85,B 0,C 180,E1 27830.639,E2 27830.639} C_VEL
LIN {X 0,Y 591.916,Z 770.746,A -85,B 0,C 180,E1 27829.22,E2 27829.22} C_VEL
LIN {X 0,Y 591.917,Z 769.015,A -85,B 0,C 180,E1 27827.803,E2 27827.803} C_VEL
LIN {X 0,Y 591.921,Z 765.396,A -85,B 0,C 180,E1 27826.371,E2 27826.371} C_VEL
LIN {X 0,Y 591.929,Z 760.459,A -85,B 0,C 180,E1 27825.078,E2 27825.078} C_VEL
LIN {X 0,Y 591.943,Z 753.024,A -85,B 0,C 180,E1 27823.678,E2 27823.678} C_VEL
LIN {X 0,Y 591.97,Z 744.606,A -85,B 0,C 180,E1 27822.486,E2 27822.486} C_VEL
LIN {X 0,Y 592.006,Z 734.861,A -85,B 0,C 180,E1 27821.397,E2 27821.397} C_VEL
LIN {X 0,Y 592.057,Z 723.044,A -85,B 0,C 180,E1 27820.361,E2 27820.361} C_VEL
LIN {X 0,Y 592.096,Z 709.939,A -85,B 0,C 180,E1 27819.477,E2 27819.477} C_VEL
LIN {X 0,Y 592.167,Z 696.441,A -85,B 0,C 180,E1 27818.789,E2 27818.789} C_VEL
LIN {X 0,Y 592.219,Z 682.157,A -85,B 0,C 180,E1 27818.263,E2 27818.263} C_VEL
LIN {X 0,Y 592.252,Z 666.494,A -85,B 0,C 180,E1 27817.896,E2 27817.896} C_VEL
LIN {X 0,Y 592.147,Z 556.923,A -85,B 0,C 180,E1 27816.535,E2 27816.535} C_VEL
LIN {X 0,Y 592.227,Z 526.003,A -85,B 0,C 180,E1 27813.387,E2 27813.387} C_VEL
LIN {X 0,Y 592.364,Z 494.442,A -85,B 0,C 180,E1 27810.097,E2 27810.097} C_VEL
LIN {X 0,Y 592.51,Z 464.426,A -85,B 0,C 180,E1 27806.904,E2 27806.904} C_VEL
LIN {X 0,Y 592.692,Z 435.013,A -85,B 0,C 180,E1 27803.704,E2 27803.704} C_VEL
LIN {X 0,Y 592.369,Z 430.728,A -85,B 0,C 180,E1 27803.214,E2 27803.214} C_VEL
LIN {X 0,Y 591.982,Z 429.151,A -85,B 0,C 180,E1 27802.966,E2 27802.966} C_VEL
LIN {X 0,Y 592.016,Z 429.055,A -85,B 0,C 180,E1 27799.944,E2 27799.944} C_VEL
LIN {X 0,Y 591.964,Z 429.055,A -85,B 0,C 180,E1 27796.819,E2 27796.819} C_VEL
LIN {X 0,Y 592.012,Z 429.054,A -85,B 0,C 180,E1 27793.819,E2 27793.819} C_VEL
LIN {X 0,Y 591.957,Z 429.055,A -85,B 0,C 180,E1 27790.667,E2 27790.667} C_VEL
LIN {X 0,Y 592.014,Z 429.054,A -85,B 0,C 180,E1 27787.666,E2 27787.666} C_VEL
LIN {X 0,Y 591.954,Z 429.055,A -85,B 0,C 180,E1 27784.594,E2 27784.594} C_VEL
LIN {X 0,Y 591.997,Z 429.055,A -85,B 0,C 180,E1 27781.637,E2 27781.637} C_VEL
LIN {X 0,Y 591.952,Z 429.055,A -85,B 0,C 180,E1 27778.538,E2 27778.538} C_VEL
LIN {X 0,Y 591.982,Z 429.055,A -85,B 0,C 180,E1 27775.658,E2 27775.658} C_VEL
LIN {X 0,Y 591.957,Z 429.054,A -85,B 0,C 180,E1 27772.428,E2 27772.428} C_VEL
LIN {X 0,Y 591.984,Z 429.055,A -85,B 0,C 180,E1 27769.566,E2 27769.566} C_VEL
LIN {X 0,Y 591.968,Z 429.054,A -85,B 0,C 180,E1 27766.436,E2 27766.436} C_VEL
LIN {X 0,Y 591.979,Z 429.055,A -85,B 0,C 180,E1 27763.561,E2 27763.561} C_VEL
LIN {X 0,Y 591.971,Z 429.052,A -85,B 0,C 180,E1 27760.309,E2 27760.309} C_VEL
LIN {X 0,Y 591.984,Z 429.055,A -85,B 0,C 180,E1 27757.448,E2 27757.448} C_VEL
LIN {X 0,Y 591.973,Z 429.05,A -85,B 0,C 180,E1 27754.144,E2 27754.144} C_VEL
LIN {X 0,Y 591.999,Z 429.054,A -85,B 0,C 180,E1 27751.233,E2 27751.233} C_VEL
LIN {X 0,Y 591.975,Z 429.051,A -85,B 0,C 180,E1 27748.005,E2 27748.005} C_VEL
LIN {X 0,Y 592.019,Z 429.052,A -85,B 0,C 180,E1 27744.975,E2 27744.975} C_VEL
LIN {X 0,Y 591.977,Z 429.052,A -85,B 0,C 180,E1 27741.814,E2 27741.814} C_VEL
LIN {X 0,Y 592.037,Z 429.052,A -85,B 0,C 180,E1 27738.716,E2 27738.716} C_VEL
LIN {X 0,Y 591.978,Z 429.051,A -85,B 0,C 180,E1 27735.578,E2 27735.578} C_VEL
LIN {X 0,Y 592.039,Z 429.051,A -85,B 0,C 180,E1 27732.485,E2 27732.485} C_VEL
LIN {X 0,Y 591.982,Z 429.05,A -85,B 0,C 180,E1 27729.332,E2 27729.332} C_VEL
LIN {X 0,Y 592.036,Z 429.049,A -85,B 0,C 180,E1 27726.205,E2 27726.205} C_VEL
LIN {X 0,Y 591.99,Z 429.052,A -85,B 0,C 180,E1 27723.098,E2 27723.098} C_VEL
LIN {X 0,Y 592.018,Z 429.045,A -85,B 0,C 180,E1 27719.807,E2 27719.807} C_VEL
LIN {X 0,Y 592.018,Z 429.054,A -85,B 0,C 180,E1 27716.611,E2 27716.611} C_VEL
LIN {X 0,Y 592,Z 429.048,A -85,B 0,C 180,E1 27713.405,E2 27713.405} C_VEL
LIN {X 0,Y 592.035,Z 429.054,A -85,B 0,C 180,E1 27710.277,E2 27710.277} C_VEL
LIN {X 0,Y 591.997,Z 429.049,A -85,B 0,C 180,E1 27707.118,E2 27707.118} C_VEL
LIN {X 0,Y 592.034,Z 429.049,A -85,B 0,C 180,E1 27703.921,E2 27703.921} C_VEL
LIN {X 0,Y 592.001,Z 429.051,A -85,B 0,C 180,E1 27700.756,E2 27700.756} C_VEL
LIN {X 0,Y 592.035,Z 429.045,A -85,B 0,C 180,E1 27697.489,E2 27697.489} C_VEL
LIN {X 0,Y 592.033,Z 429.055,A -85,B 0,C 180,E1 27694.169,E2 27694.169} C_VEL
LIN {X 0,Y 592.006,Z 429.049,A -85,B 0,C 180,E1 27690.895,E2 27690.895} C_VEL
LIN {X 0,Y 592.03,Z 429.051,A -85,B 0,C 180,E1 27687.746,E2 27687.746} C_VEL
LIN {X 0,Y 592.007,Z 429.05,A -85,B 0,C 180,E1 27684.599,E2 27684.599} C_VEL
LIN {X 0,Y 592.029,Z 429.048,A -85,B 0,C 180,E1 27681.439,E2 27681.439} C_VEL
LIN {X 0,Y 592.013,Z 429.052,A -85,B 0,C 180,E1 27678.285,E2 27678.285} C_VEL
LIN {X 0,Y 592.035,Z 429.044,A -85,B 0,C 180,E1 27674.958,E2 27674.958} C_VEL
LIN {X 0,Y 592.033,Z 429.055,A -85,B 0,C 180,E1 27671.714,E2 27671.714} C_VEL
LIN {X 0,Y 592.019,Z 429.048,A -85,B 0,C 180,E1 27668.551,E2 27668.551} C_VEL
LIN {X 0,Y 592.023,Z 429.051,A -85,B 0,C 180,E1 27665.34,E2 27665.34} C_VEL
LIN {X 0,Y 592.017,Z 429.049,A -85,B 0,C 180,E1 27662.141,E2 27662.141} C_VEL
LIN {X 0,Y 592.054,Z 429.221,A -85,B 0,C 180,E1 27660.539,E2 27660.539} C_VEL
LIN {X 0,Y 593.397,Z 433.886,A -85,B 0,C 180,E1 27660.085,E2 27660.085} C_VEL
LIN {X 0,Y 593.111,Z 478.781,A -85,B 0,C 180,E1 27656.967,E2 27656.967} C_VEL
LIN {X 0,Y 592.824,Z 526.04,A -85,B 0,C 180,E1 27653.772,E2 27653.772} C_VEL
LIN {X 0,Y 592.867,Z 539.114,A -85,B 0,C 180,E1 27652.926,E2 27652.926} C_VEL
LIN {X 0,Y 593.11,Z 550.611,A -85,B 0,C 180,E1 27652.765,E2 27652.765} C_VEL
LIN {X 0,Y 592.846,Z 748.31,A -85,B 0,C 180,E1 27650.227,E2 27650.227} C_VEL
LIN {X 0,Y 592.745,Z 767.302,A -85,B 0,C 180,E1 27649.798,E2 27649.798} C_VEL
LIN {X 0,Y 592.662,Z 785.402,A -85,B 0,C 180,E1 27649.207,E2 27649.207} C_VEL
LIN {X 0,Y 592.55,Z 803.052,A -85,B 0,C 180,E1 27648.445,E2 27648.445} C_VEL
LIN {X 0,Y 592.459,Z 819.696,A -85,B 0,C 180,E1 27647.538,E2 27647.538} C_VEL
LIN {X 0,Y 592.342,Z 835.636,A -85,B 0,C 180,E1 27646.474,E2 27646.474} C_VEL
LIN {X 0,Y 592.23,Z 850.561,A -85,B 0,C 180,E1 27645.271,E2 27645.271} C_VEL
LIN {X 0,Y 592.131,Z 864.018,A -85,B 0,C 180,E1 27643.973,E2 27643.973} C_VEL
LIN {X 0,Y 592.058,Z 876.908,A -85,B 0,C 180,E1 27642.484,E2 27642.484} C_VEL
LIN {X 0,Y 591.998,Z 888.225,A -85,B 0,C 180,E1 27640.904,E2 27640.904} C_VEL
LIN {X 0,Y 591.954,Z 897.99,A -85,B 0,C 180,E1 27639.234,E2 27639.234} C_VEL
LIN {X 0,Y 591.935,Z 905.772,A -85,B 0,C 180,E1 27637.571,E2 27637.571} C_VEL
LIN {X 0,Y 591.913,Z 912.262,A -85,B 0,C 180,E1 27635.767,E2 27635.767} C_VEL
LIN {X 0,Y 591.919,Z 916.873,A -85,B 0,C 180,E1 27633.971,E2 27633.971} C_VEL
LIN {X 0,Y 591.917,Z 919.788,A -85,B 0,C 180,E1 27632.13,E2 27632.13} C_VEL
LIN {X 0,Y 591.907,Z 920.94,A -85,B 0,C 180,E1 27630.291,E2 27630.291} C_VEL
LIN {X 0,Y 591.915,Z 920.349,A -85,B 0,C 180,E1 27628.451,E2 27628.451} C_VEL
LIN {X 0,Y 591.907,Z 918.006,A -85,B 0,C 180,E1 27626.611,E2 27626.611} C_VEL
LIN {X 0,Y 591.912,Z 914.098,A -85,B 0,C 180,E1 27624.864,E2 27624.864} C_VEL
LIN {X 0,Y 591.928,Z 908.468,A -85,B 0,C 180,E1 27623.112,E2 27623.112} C_VEL
LIN {X 0,Y 591.94,Z 901.424,A -85,B 0,C 180,E1 27621.452,E2 27621.452} C_VEL
LIN {X 0,Y 591.977,Z 892.511,A -85,B 0,C 180,E1 27619.785,E2 27619.785} C_VEL
LIN {X 0,Y 592.024,Z 882.147,A -85,B 0,C 180,E1 27618.208,E2 27618.208} C_VEL
LIN {X 0,Y 592.093,Z 870.348,A -85,B 0,C 180,E1 27616.723,E2 27616.723} C_VEL
LIN {X 0,Y 592.193,Z 856.581,A -85,B 0,C 180,E1 27615.28,E2 27615.28} C_VEL
LIN {X 0,Y 592.305,Z 841.597,A -85,B 0,C 180,E1 27613.978,E2 27613.978} C_VEL
LIN {X 0,Y 592.421,Z 825.421,A -85,B 0,C 180,E1 27612.821,E2 27612.821} C_VEL
LIN {X 0,Y 592.514,Z 809.037,A -85,B 0,C 180,E1 27611.86,E2 27611.86} C_VEL
LIN {X 0,Y 592.649,Z 792.227,A -85,B 0,C 180,E1 27611.066,E2 27611.066} C_VEL
LIN {X 0,Y 592.72,Z 774.059,A -85,B 0,C 180,E1 27610.402,E2 27610.402} C_VEL
LIN {X 0,Y 592.816,Z 755.473,A -85,B 0,C 180,E1 27609.914,E2 27609.914} C_VEL
LIN {X 0,Y 592.883,Z 735.648,A -85,B 0,C 180,E1 27609.588,E2 27609.588} C_VEL
LIN {X 0,Y 592.952,Z 539.717,A -85,B 0,C 180,E1 27607.089,E2 27607.089} C_VEL
LIN {X 0,Y 592.789,Z 537.072,A -85,B 0,C 180,E1 27606.964,E2 27606.964} C_VEL
LIN {X 0,Y 593.045,Z 489.105,A -85,B 0,C 180,E1 27603.738,E2 27603.738} C_VEL
LIN {X 0,Y 593.332,Z 443.662,A -85,B 0,C 180,E1 27600.602,E2 27600.602} C_VEL
LIN {X 0,Y 593.231,Z 432.971,A -85,B 0,C 180,E1 27599.841,E2 27599.841} C_VEL
LIN {X 0,Y 592.053,Z 429.223,A -85,B 0,C 180,E1 27599.461,E2 27599.461} C_VEL
LIN {X 0,Y 592.029,Z 429.055,A -85,B 0,C 180,E1 27596.129,E2 27596.129} C_VEL
LIN {X 0,Y 592.023,Z 429.048,A -85,B 0,C 180,E1 27592.859,E2 27592.859} C_VEL
LIN {X 0,Y 592.017,Z 429.05,A -85,B 0,C 180,E1 27589.696,E2 27589.696} C_VEL
LIN {X 0,Y 592.022,Z 429.049,A -85,B 0,C 180,E1 27586.571,E2 27586.571} C_VEL
LIN {X 0,Y 592.017,Z 429.049,A -85,B 0,C 180,E1 27583.423,E2 27583.423} C_VEL
LIN {X 0,Y 592.028,Z 429.053,A -85,B 0,C 180,E1 27580.177,E2 27580.177} C_VEL
LIN {X 0,Y 592.035,Z 429.045,A -85,B 0,C 180,E1 27576.821,E2 27576.821} C_VEL
LIN {X 0,Y 592.02,Z 429.052,A -85,B 0,C 180,E1 27573.523,E2 27573.523} C_VEL
LIN {X 0,Y 592.024,Z 429.048,A -85,B 0,C 180,E1 27570.33,E2 27570.33} C_VEL
LIN {X 0,Y 592.015,Z 429.049,A -85,B 0,C 180,E1 27567.12,E2 27567.12} C_VEL
LIN {X 0,Y 592.026,Z 429.051,A -85,B 0,C 180,E1 27563.912,E2 27563.912} C_VEL
LIN {X 0,Y 592.024,Z 429.046,A -85,B 0,C 180,E1 27560.669,E2 27560.669} C_VEL
LIN {X 0,Y 592.025,Z 429.053,A -85,B 0,C 180,E1 27557.292,E2 27557.292} C_VEL
LIN {X 0,Y 592.028,Z 429.045,A -85,B 0,C 180,E1 27554.075,E2 27554.075} C_VEL
LIN {X 0,Y 592.013,Z 429.05,A -85,B 0,C 180,E1 27550.904,E2 27550.904} C_VEL
LIN {X 0,Y 592.025,Z 429.049,A -85,B 0,C 180,E1 27547.765,E2 27547.765} C_VEL
LIN {X 0,Y 592.013,Z 429.047,A -85,B 0,C 180,E1 27544.553,E2 27544.553} C_VEL
LIN {X 0,Y 592.03,Z 429.053,A -85,B 0,C 180,E1 27541.355,E2 27541.355} C_VEL
LIN {X 0,Y 592.03,Z 429.045,A -85,B 0,C 180,E1 27538.064,E2 27538.064} C_VEL
LIN {X 0,Y 592.02,Z 429.052,A -85,B 0,C 180,E1 27534.767,E2 27534.767} C_VEL
LIN {X 0,Y 592.028,Z 429.047,A -85,B 0,C 180,E1 27531.551,E2 27531.551} C_VEL
LIN {X 0,Y 592.015,Z 429.046,A -85,B 0,C 180,E1 27530.116,E2 27530.116} C_VEL
LIN {X 0,Y 591.064,Z 429.168,A -85,B 0,C 180,E1 27529.37,E2 27529.37} C_VEL
LIN {X 0,Y 584.561,Z 429.988,A -85,B 0,C 180,E1 27527.224,E2 27527.224} C_VEL
LIN {X 0,Y 584.09,Z 430.041,A -85,B 0,C 180,E1 27526.734,E2 27526.734} C_VEL
LIN {X 0,Y 584.094,Z 430.035,A -85,B 0,C 180,E1 27523.458,E2 27523.458} C_VEL
LIN {X 0,Y 584.071,Z 430.039,A -85,B 0,C 180,E1 27520.187,E2 27520.187} C_VEL
LIN {X 0,Y 584.088,Z 430.04,A -85,B 0,C 180,E1 27517.027,E2 27517.027} C_VEL
LIN {X 0,Y 584.076,Z 430.037,A -85,B 0,C 180,E1 27513.769,E2 27513.769} C_VEL
LIN {X 0,Y 584.09,Z 430.043,A -85,B 0,C 180,E1 27510.413,E2 27510.413} C_VEL
LIN {X 0,Y 584.095,Z 430.035,A -85,B 0,C 180,E1 27507.136,E2 27507.136} C_VEL
LIN {X 0,Y 584.071,Z 430.041,A -85,B 0,C 180,E1 27503.902,E2 27503.902} C_VEL
LIN {X 0,Y 584.09,Z 430.042,A -85,B 0,C 180,E1 27500.691,E2 27500.691} C_VEL
LIN {X 0,Y 584.071,Z 430.043,A -85,B 0,C 180,E1 27497.546,E2 27497.546} C_VEL
LIN {X 0,Y 584.135,Z 430.356,A -85,B 0,C 180,E1 27497.175,E2 27497.175} C_VEL
LIN {X 0,Y 585.103,Z 435,A -85,B 0,C 180,E1 27496.574,E2 27496.574} C_VEL
LIN {X 0,Y 584.838,Z 464.197,A -85,B 0,C 180,E1 27493.351,E2 27493.351} C_VEL
LIN {X 0,Y 584.593,Z 494.338,A -85,B 0,C 180,E1 27490.1,E2 27490.1} C_VEL
LIN {X 0,Y 584.402,Z 525.517,A -85,B 0,C 180,E1 27486.802,E2 27486.802} C_VEL
LIN {X 0,Y 584.211,Z 556.218,A -85,B 0,C 180,E1 27483.618,E2 27483.618} C_VEL
LIN {X 0,Y 584.393,Z 558.209,A -85,B 0,C 180,E1 27483.529,E2 27483.529} C_VEL
LIN {X 0,Y 584.389,Z 668.472,A -85,B 0,C 180,E1 27482.141,E2 27482.141} C_VEL
LIN {X 0,Y 584.363,Z 683.257,A -85,B 0,C 180,E1 27481.773,E2 27481.773} C_VEL
LIN {X 0,Y 584.29,Z 698.055,A -85,B 0,C 180,E1 27481.201,E2 27481.201} C_VEL
LIN {X 0,Y 584.178,Z 711.098,A -85,B 0,C 180,E1 27480.506,E2 27480.506} C_VEL
LIN {X 0,Y 584.122,Z 723.443,A -85,B 0,C 180,E1 27479.649,E2 27479.649} C_VEL
LIN {X 0,Y 584.052,Z 735.47,A -85,B 0,C 180,E1 27478.571,E2 27478.571} C_VEL
LIN {X 0,Y 583.992,Z 745.85,A -85,B 0,C 180,E1 27477.368,E2 27477.368} C_VEL
LIN {X 0,Y 583.952,Z 754.257,A -85,B 0,C 180,E1 27476.106,E2 27476.106} C_VEL
LIN {X 0,Y 583.932,Z 760.885,A -85,B 0,C 180,E1 27474.804,E2 27474.804} C_VEL
LIN {X 0,Y 583.92,Z 766.28,A -85,B 0,C 180,E1 27473.3,E2 27473.3} C_VEL
LIN {X 0,Y 583.916,Z 769.541,A -85,B 0,C 180,E1 27471.813,E2 27471.813} C_VEL
LIN {X 0,Y 583.918,Z 770.894,A -85,B 0,C 180,E1 27470.445,E2 27470.445} C_VEL
LIN {X 0,Y 583.915,Z 770.521,A -85,B 0,C 180,E1 27468.883,E2 27468.883} C_VEL
LIN {X 0,Y 583.918,Z 768.327,A -85,B 0,C 180,E1 27467.437,E2 27467.437} C_VEL
LIN {X 0,Y 583.923,Z 764.352,A -85,B 0,C 180,E1 27466.003,E2 27466.003} C_VEL
LIN {X 0,Y 583.939,Z 758.441,A -85,B 0,C 180,E1 27464.578,E2 27464.578} C_VEL
LIN {X 0,Y 583.967,Z 750.923,A -85,B 0,C 180,E1 27463.264,E2 27463.264} C_VEL
LIN {X 0,Y 584.011,Z 741.954,A -85,B 0,C 180,E1 27462.056,E2 27462.056} C_VEL
LIN {X 0,Y 584.077,Z 731.516,A -85,B 0,C 180,E1 27460.954,E2 27460.954} C_VEL
LIN {X 0,Y 584.154,Z 719.379,A -85,B 0,C 180,E1 27459.955,E2 27459.955} C_VEL
LIN {X 0,Y 584.225,Z 706.876,A -85,B 0,C 180,E1 27459.158,E2 27459.158} C_VEL
LIN {X 0,Y 584.317,Z 693.571,A -85,B 0,C 180,E1 27458.512,E2 27458.512} C_VEL
LIN {X 0,Y 584.388,Z 678.026,A -85,B 0,C 180,E1 27457.984,E2 27457.984} C_VEL
LIN {X 0,Y 584.433,Z 662.828,A -85,B 0,C 180,E1 27457.678,E2 27457.678} C_VEL
LIN {X 0,Y 584.316,Z 557.51,A -85,B 0,C 180,E1 27456.367,E2 27456.367} C_VEL
LIN {X 0,Y 584.234,Z 555.124,A -85,B 0,C 180,E1 27456.189,E2 27456.189} C_VEL
LIN {X 0,Y 584.375,Z 523.945,A -85,B 0,C 180,E1 27452.942,E2 27452.942} C_VEL
LIN {X 0,Y 584.614,Z 493.357,A -85,B 0,C 180,E1 27449.706,E2 27449.706} C_VEL
LIN {X 0,Y 584.838,Z 463.394,A -85,B 0,C 180,E1 27446.471,E2 27446.471} C_VEL
LIN {X 0,Y 585.105,Z 434.479,A -85,B 0,C 180,E1 27443.278,E2 27443.278} C_VEL
LIN {X 0,Y 584.04,Z 430.147,A -85,B 0,C 180,E1 27442.672,E2 27442.672} C_VEL
LIN {X 0,Y 584.091,Z 430.045,A -85,B 0,C 180,E1 27439.545,E2 27439.545} C_VEL
LIN {X 0,Y 584.023,Z 430.043,A -85,B 0,C 180,E1 27436.516,E2 27436.516} C_VEL
LIN {X 0,Y 584.079,Z 430.044,A -85,B 0,C 180,E1 27433.388,E2 27433.388} C_VEL
LIN {X 0,Y 584.018,Z 430.043,A -85,B 0,C 180,E1 27430.393,E2 27430.393} C_VEL
LIN {X 0,Y 584.071,Z 430.039,A -85,B 0,C 180,E1 27427.239,E2 27427.239} C_VEL
LIN {X 0,Y 584.016,Z 430.044,A -85,B 0,C 180,E1 27424.223,E2 27424.223} C_VEL
LIN {X 0,Y 584.052,Z 430.045,A -85,B 0,C 180,E1 27421.022,E2 27421.022} C_VEL
LIN {X 0,Y 584.011,Z 430.044,A -85,B 0,C 180,E1 27418.123,E2 27418.123} C_VEL
LIN {X 0,Y 584.066,Z 430.043,A -85,B 0,C 180,E1 27415.006,E2 27415.006} C_VEL
LIN {X 0,Y 584.015,Z 430.043,A -85,B 0,C 180,E1 27412.075,E2 27412.075} C_VEL
LIN {X 0,Y 584.072,Z 430.041,A -85,B 0,C 180,E1 27408.901,E2 27408.901} C_VEL
LIN {X 0,Y 584.019,Z 430.043,A -85,B 0,C 180,E1 27405.966,E2 27405.966} C_VEL
LIN {X 0,Y 584.079,Z 430.04,A -85,B 0,C 180,E1 27402.813,E2 27402.813} C_VEL
LIN {X 0,Y 584.025,Z 430.042,A -85,B 0,C 180,E1 27399.814,E2 27399.814} C_VEL
LIN {X 0,Y 584.068,Z 430.04,A -85,B 0,C 180,E1 27396.594,E2 27396.594} C_VEL
LIN {X 0,Y 584.029,Z 430.039,A -85,B 0,C 180,E1 27393.69,E2 27393.69} C_VEL
LIN {X 0,Y 584.082,Z 430.04,A -85,B 0,C 180,E1 27390.559,E2 27390.559} C_VEL
LIN {X 0,Y 584.036,Z 430.041,A -85,B 0,C 180,E1 27387.525,E2 27387.525} C_VEL
LIN {X 0,Y 584.064,Z 430.039,A -85,B 0,C 180,E1 27384.259,E2 27384.259} C_VEL
LIN {X 0,Y 584.047,Z 430.043,A -85,B 0,C 180,E1 27381.281,E2 27381.281} C_VEL
LIN {X 0,Y 584.051,Z 430.035,A -85,B 0,C 180,E1 27377.948,E2 27377.948} C_VEL
LIN {X 0,Y 584.076,Z 430.042,A -85,B 0,C 180,E1 27374.879,E2 27374.879} C_VEL
LIN {X 0,Y 584.045,Z 430.039,A -85,B 0,C 180,E1 27371.655,E2 27371.655} C_VEL
LIN {X 0,Y 584.097,Z 430.039,A -85,B 0,C 180,E1 27368.565,E2 27368.565} C_VEL
LIN {X 0,Y 584.046,Z 430.04,A -85,B 0,C 180,E1 27365.403,E2 27365.403} C_VEL
LIN {X 0,Y 584.099,Z 430.037,A -85,B 0,C 180,E1 27362.257,E2 27362.257} C_VEL
LIN {X 0,Y 584.05,Z 430.037,A -85,B 0,C 180,E1 27359.117,E2 27359.117} C_VEL
LIN {X 0,Y 584.092,Z 430.036,A -85,B 0,C 180,E1 27355.877,E2 27355.877} C_VEL
LIN {X 0,Y 584.067,Z 430.04,A -85,B 0,C 180,E1 27352.722,E2 27352.722} C_VEL
LIN {X 0,Y 584.062,Z 430.038,A -85,B 0,C 180,E1 27349.346,E2 27349.346} C_VEL
LIN {X 0,Y 584.098,Z 430.039,A -85,B 0,C 180,E1 27346.134,E2 27346.134} C_VEL
LIN {X 0,Y 584.059,Z 430.038,A -85,B 0,C 180,E1 27342.978,E2 27342.978} C_VEL
LIN {X 0,Y 584.096,Z 430.035,A -85,B 0,C 180,E1 27339.731,E2 27339.731} C_VEL
LIN {X 0,Y 584.072,Z 430.041,A -85,B 0,C 180,E1 27336.493,E2 27336.493} C_VEL
LIN {X 0,Y 584.076,Z 430.034,A -85,B 0,C 180,E1 27333.111,E2 27333.111} C_VEL
LIN {X 0,Y 584.096,Z 430.041,A -85,B 0,C 180,E1 27329.897,E2 27329.897} C_VEL
LIN {X 0,Y 584.068,Z 430.038,A -85,B 0,C 180,E1 27326.658,E2 27326.658} C_VEL
LIN {X 0,Y 584.093,Z 430.036,A -85,B 0,C 180,E1 27323.403,E2 27323.403} C_VEL
LIN {X 0,Y 584.08,Z 430.041,A -85,B 0,C 180,E1 27320.191,E2 27320.191} C_VEL
LIN {X 0,Y 584.082,Z 430.036,A -85,B 0,C 180,E1 27316.785,E2 27316.785} C_VEL
LIN {X 0,Y 584.091,Z 430.042,A -85,B 0,C 180,E1 27313.606,E2 27313.606} C_VEL
LIN {X 0,Y 584.075,Z 430.04,A -85,B 0,C 180,E1 27310.323,E2 27310.323} C_VEL
LIN {X 0,Y 584.089,Z 430.037,A -85,B 0,C 180,E1 27307.054,E2 27307.054} C_VEL
LIN {X 0,Y 584.094,Z 430.045,A -85,B 0,C 180,E1 27303.702,E2 27303.702} C_VEL
LIN {X 0,Y 584.113,Z 430.224,A -85,B 0,C 180,E1 27300.926,E2 27300.926} C_VEL
LIN {X 0,Y 585.674,Z 435.003,A -85,B 0,C 180,E1 27300.443,E2 27300.443} C_VEL
LIN {X 0,Y 586.143,Z 437.036,A -85,B 0,C 180,E1 27300.27,E2 27300.27} C_VEL
LIN {X 0,Y 585.709,Z 481.932,A -85,B 0,C 180,E1 27297.116,E2 27297.116} C_VEL
LIN {X 0,Y 585.299,Z 528.272,A -85,B 0,C 180,E1 27293.945,E2 27293.945} C_VEL
LIN {X 0,Y 585.341,Z 539.263,A -85,B 0,C 180,E1 27293.235,E2 27293.235} C_VEL
LIN {X 0,Y 585.744,Z 545.013,A -85,B 0,C 180,E1 27293.14,E2 27293.14} C_VEL
LIN {X 0,Y 585.336,Z 748.31,A -85,B 0,C 180,E1 27290.498,E2 27290.498} C_VEL
LIN {X 0,Y 585.198,Z 767.301,A -85,B 0,C 180,E1 27290.064,E2 27290.064} C_VEL
LIN {X 0,Y 585.066,Z 785.4,A -85,B 0,C 180,E1 27289.466,E2 27289.466} C_VEL
LIN {X 0,Y 584.901,Z 803.048,A -85,B 0,C 180,E1 27288.695,E2 27288.695} C_VEL
LIN {X 0,Y 584.738,Z 820.22,A -85,B 0,C 180,E1 27287.744,E2 27287.744} C_VEL
LIN {X 0,Y 584.56,Z 836.234,A -85,B 0,C 180,E1 27286.654,E2 27286.654} C_VEL
LIN {X 0,Y 584.393,Z 851.098,A -85,B 0,C 180,E1 27285.431,E2 27285.431} C_VEL
LIN {X 0,Y 584.241,Z 864.944,A -85,B 0,C 180,E1 27284.065,E2 27284.065} C_VEL
LIN {X 0,Y 584.129,Z 877.683,A -85,B 0,C 180,E1 27282.556,E2 27282.556} C_VEL
LIN {X 0,Y 584.04,Z 888.865,A -85,B 0,C 180,E1 27280.955,E2 27280.955} C_VEL
LIN {X 0,Y 583.976,Z 898.508,A -85,B 0,C 180,E1 27279.262,E2 27279.262} C_VEL
LIN {X 0,Y 583.942,Z 906.402,A -85,B 0,C 180,E1 27277.521,E2 27277.521} C_VEL
LIN {X 0,Y 583.917,Z 912.41,A -85,B 0,C 180,E1 27275.799,E2 27275.799} C_VEL
LIN {X 0,Y 583.919,Z 916.874,A -85,B 0,C 180,E1 27274.026,E2 27274.026} C_VEL
LIN {X 0,Y 583.917,Z 919.789,A -85,B 0,C 180,E1 27272.159,E2 27272.159} C_VEL
LIN {X 0,Y 583.907,Z 920.94,A -85,B 0,C 180,E1 27270.295,E2 27270.295} C_VEL
LIN {X 0,Y 583.915,Z 920.349,A -85,B 0,C 180,E1 27268.43,E2 27268.43} C_VEL
LIN {X 0,Y 583.907,Z 918.006,A -85,B 0,C 180,E1 27266.564,E2 27266.564} C_VEL
LIN {X 0,Y 583.916,Z 914.098,A -85,B 0,C 180,E1 27264.793,E2 27264.793} C_VEL
LIN {X 0,Y 583.934,Z 908.469,A -85,B 0,C 180,E1 27263.017,E2 27263.017} C_VEL
LIN {X 0,Y 583.955,Z 901.425,A -85,B 0,C 180,E1 27261.334,E2 27261.334} C_VEL
LIN {X 0,Y 584.016,Z 892.512,A -85,B 0,C 180,E1 27259.644,E2 27259.644} C_VEL
LIN {X 0,Y 584.086,Z 882.148,A -85,B 0,C 180,E1 27258.046,E2 27258.046} C_VEL
LIN {X 0,Y 584.194,Z 870.348,A -85,B 0,C 180,E1 27256.54,E2 27256.54} C_VEL
LIN {X 0,Y 584.342,Z 856.58,A -85,B 0,C 180,E1 27255.077,E2 27255.077} C_VEL
LIN {X 0,Y 584.508,Z 841.599,A -85,B 0,C 180,E1 27253.759,E2 27253.759} C_VEL
LIN {X 0,Y 584.685,Z 825.424,A -85,B 0,C 180,E1 27252.587,E2 27252.587} C_VEL
LIN {X 0,Y 584.839,Z 808.667,A -85,B 0,C 180,E1 27251.594,E2 27251.594} C_VEL
LIN {X 0,Y 585.032,Z 791.8,A -85,B 0,C 180,E1 27250.792,E2 27250.792} C_VEL
LIN {X 0,Y 585.156,Z 773.738,A -85,B 0,C 180,E1 27250.128,E2 27250.128} C_VEL
LIN {X 0,Y 585.295,Z 755.311,A -85,B 0,C 180,E1 27249.641,E2 27249.641} C_VEL
LIN {X 0,Y 585.386,Z 735.442,A -85,B 0,C 180,E1 27249.312,E2 27249.312} C_VEL
LIN {X 0,Y 585.577,Z 540.776,A -85,B 0,C 180,E1 27246.797,E2 27246.797} C_VEL
LIN {X 0,Y 585.248,Z 537.884,A -85,B 0,C 180,E1 27246.703,E2 27246.703} C_VEL
LIN {X 0,Y 585.633,Z 490.282,A -85,B 0,C 180,E1 27243.461,E2 27243.461} C_VEL
LIN {X 0,Y 586.068,Z 444.641,A -85,B 0,C 180,E1 27240.271,E2 27240.271} C_VEL
LIN {X 0,Y 585.919,Z 435.583,A -85,B 0,C 180,E1 27239.613,E2 27239.613} C_VEL
LIN {X 0,Y 584.134,Z 430.349,A -85,B 0,C 180,E1 27239.102,E2 27239.102} C_VEL
LIN {X 0,Y 584.079,Z 430.04,A -85,B 0,C 180,E1 27237.833,E2 27237.833} C_VEL
LIN {X 0,Y 584.085,Z 430.043,A -85,B 0,C 180,E1 27234.571,E2 27234.571} C_VEL
LIN {X 0,Y 584.09,Z 430.035,A -85,B 0,C 180,E1 27231.315,E2 27231.315} C_VEL
LIN {X 0,Y 584.092,Z 430.042,A -85,B 0,C 180,E1 27227.981,E2 27227.981} C_VEL
LIN {X 0,Y 584.086,Z 430.036,A -85,B 0,C 180,E1 27224.714,E2 27224.714} C_VEL
LIN {X 0,Y 584.078,Z 430.039,A -85,B 0,C 180,E1 27221.49,E2 27221.49} C_VEL
LIN {X 0,Y 584.086,Z 430.039,A -85,B 0,C 180,E1 27218.212,E2 27218.212} C_VEL
LIN {X 0,Y 584.09,Z 430.034,A -85,B 0,C 180,E1 27214.919,E2 27214.919} C_VEL
LIN {X 0,Y 584.087,Z 430.042,A -85,B 0,C 180,E1 27211.589,E2 27211.589} C_VEL
LIN {X 0,Y 584.086,Z 430.036,A -85,B 0,C 180,E1 27208.306,E2 27208.306} C_VEL
LIN {X 0,Y 584.076,Z 430.037,A -85,B 0,C 180,E1 27205.099,E2 27205.099} C_VEL
LIN {X 0,Y 584.086,Z 430.04,A -85,B 0,C 180,E1 27201.904,E2 27201.904} C_VEL
LIN {X 0,Y 584.083,Z 430.034,A -85,B 0,C 180,E1 27198.67,E2 27198.67} C_VEL
LIN {X 0,Y 584.088,Z 430.04,A -85,B 0,C 180,E1 27195.285,E2 27195.285} C_VEL
LIN {X 0,Y 584.09,Z 430.036,A -85,B 0,C 180,E1 27192.054,E2 27192.054} C_VEL
LIN {X 0,Y 584.075,Z 430.039,A -85,B 0,C 180,E1 27188.863,E2 27188.863} C_VEL
LIN {X 0,Y 584.086,Z 430.038,A -85,B 0,C 180,E1 27185.698,E2 27185.698} C_VEL
LIN {X 0,Y 584.076,Z 430.037,A -85,B 0,C 180,E1 27182.453,E2 27182.453} C_VEL
LIN {X 0,Y 584.096,Z 430.042,A -85,B 0,C 180,E1 27179.117,E2 27179.117} C_VEL
LIN {X 0,Y 584.093,Z 430.034,A -85,B 0,C 180,E1 27175.779,E2 27175.779} C_VEL
LIN {X 0,Y 584.073,Z 430.04,A -85,B 0,C 180,E1 27172.524,E2 27172.524} C_VEL
LIN {X 0,Y 584.088,Z 430.038,A -85,B 0,C 180,E1 27169.292,E2 27169.292} C_VEL
LIN {X 0,Y 584.09,Z 430.041,A -85,B 0,C 180,E1 27166.734,E2 27166.734} C_VEL
LIN {X 0,Y 583.063,Z 430.164,A -85,B 0,C 180,E1 27165.978,E2 27165.978} C_VEL
LIN {X 0,Y 576.678,Z 430.959,A -85,B 0,C 180,E1 27163.857,E2 27163.857} C_VEL
LIN {X 0,Y 576.151,Z 431.027,A -85,B 0,C 180,E1 27163.306,E2 27163.306} C_VEL
LIN {X 0,Y 576.132,Z 431.027,A -85,B 0,C 180,E1 27160.114,E2 27160.114} C_VEL
LIN {X 0,Y 576.154,Z 431.03,A -85,B 0,C 180,E1 27156.891,E2 27156.891} C_VEL
LIN {X 0,Y 576.149,Z 431.024,A -85,B 0,C 180,E1 27153.569,E2 27153.569} C_VEL
LIN {X 0,Y 576.137,Z 431.031,A -85,B 0,C 180,E1 27150.195,E2 27150.195} C_VEL
LIN {X 0,Y 576.151,Z 431.027,A -85,B 0,C 180,E1 27146.951,E2 27146.951} C_VEL
LIN {X 0,Y 576.131,Z 431.029,A -85,B 0,C 180,E1 27143.715,E2 27143.715} C_VEL
LIN {X 0,Y 576.156,Z 431.032,A -85,B 0,C 180,E1 27140.4,E2 27140.4} C_VEL
LIN {X 0,Y 576.171,Z 431.299,A -85,B 0,C 180,E1 27137.511,E2 27137.511} C_VEL
LIN {X 0,Y 577.576,Z 437.296,A -85,B 0,C 180,E1 27136.722,E2 27136.722} C_VEL
LIN {X 0,Y 577.157,Z 465.022,A -85,B 0,C 180,E1 27133.59,E2 27133.59} C_VEL
LIN {X 0,Y 576.831,Z 495.117,A -85,B 0,C 180,E1 27130.298,E2 27130.298} C_VEL
LIN {X 0,Y 576.574,Z 525.918,A -85,B 0,C 180,E1 27126.995,E2 27126.995} C_VEL
LIN {X 0,Y 576.323,Z 556.36,A -85,B 0,C 180,E1 27123.796,E2 27123.796} C_VEL
LIN {X 0,Y 576.615,Z 559.04,A -85,B 0,C 180,E1 27123.706,E2 27123.706} C_VEL
LIN {X 0,Y 576.566,Z 668.421,A -85,B 0,C 180,E1 27122.31,E2 27122.31} C_VEL
LIN {X 0,Y 576.522,Z 683.304,A -85,B 0,C 180,E1 27121.935,E2 27121.935} C_VEL
LIN {X 0,Y 576.424,Z 698.038,A -85,B 0,C 180,E1 27121.357,E2 27121.357} C_VEL
LIN {X 0,Y 576.279,Z 711.637,A -85,B 0,C 180,E1 27120.618,E2 27120.618} C_VEL
LIN {X 0,Y 576.192,Z 723.795,A -85,B 0,C 180,E1 27119.755,E2 27119.755} C_VEL
LIN {X 0,Y 576.1,Z 735.596,A -85,B 0,C 180,E1 27118.678,E2 27118.678} C_VEL
LIN {X 0,Y 576.019,Z 745.639,A -85,B 0,C 180,E1 27117.498,E2 27117.498} C_VEL
LIN {X 0,Y 575.969,Z 753.786,A -85,B 0,C 180,E1 27116.274,E2 27116.274} C_VEL
LIN {X 0,Y 575.938,Z 760.533,A -85,B 0,C 180,E1 27114.952,E2 27114.952} C_VEL
LIN {X 0,Y 575.922,Z 765.713,A -85,B 0,C 180,E1 27113.534,E2 27113.534} C_VEL
LIN {X 0,Y 575.919,Z 769.075,A -85,B 0,C 180,E1 27112.131,E2 27112.131} C_VEL
LIN {X 0,Y 575.917,Z 770.865,A -85,B 0,C 180,E1 27110.53,E2 27110.53} C_VEL
LIN {X 0,Y 575.915,Z 770.575,A -85,B 0,C 180,E1 27108.945,E2 27108.945} C_VEL
LIN {X 0,Y 575.919,Z 768.483,A -85,B 0,C 180,E1 27107.478,E2 27107.478} C_VEL
LIN {X 0,Y 575.925,Z 764.621,A -85,B 0,C 180,E1 27106.024,E2 27106.024} C_VEL
LIN {X 0,Y 575.944,Z 758.793,A -85,B 0,C 180,E1 27104.579,E2 27104.579} C_VEL
LIN {X 0,Y 575.982,Z 751.408,A -85,B 0,C 180,E1 27103.246,E2 27103.246} C_VEL
LIN {X 0,Y 576.042,Z 742.594,A -85,B 0,C 180,E1 27102.022,E2 27102.022} C_VEL
LIN {X 0,Y 576.133,Z 731.778,A -85,B 0,C 180,E1 27100.853,E2 27100.853} C_VEL
LIN {X 0,Y 576.235,Z 719.705,A -85,B 0,C 180,E1 27099.841,E2 27099.841} C_VEL
LIN {X 0,Y 576.335,Z 707.308,A -85,B 0,C 180,E1 27099.033,E2 27099.033} C_VEL
LIN {X 0,Y 576.454,Z 694.135,A -85,B 0,C 180,E1 27098.378,E2 27098.378} C_VEL
LIN {X 0,Y 576.543,Z 679.271,A -85,B 0,C 180,E1 27097.856,E2 27097.856} C_VEL
LIN {X 0,Y 576.611,Z 664.611,A -85,B 0,C 180,E1 27097.535,E2 27097.535} C_VEL
LIN {X 0,Y 576.544,Z 558.358,A -85,B 0,C 180,E1 27096.194,E2 27096.194} C_VEL
LIN {X 0,Y 576.36,Z 556.471,A -85,B 0,C 180,E1 27096.124,E2 27096.124} C_VEL
LIN {X 0,Y 576.545,Z 525.621,A -85,B 0,C 180,E1 27092.883,E2 27092.883} C_VEL
LIN {X 0,Y 576.851,Z 495.027,A -85,B 0,C 180,E1 27089.603,E2 27089.603} C_VEL
LIN {X 0,Y 577.156,Z 465.061,A -85,B 0,C 180,E1 27086.325,E2 27086.325} C_VEL
LIN {X 0,Y 577.549,Z 436.763,A -85,B 0,C 180,E1 27083.139,E2 27083.139} C_VEL
LIN {X 0,Y 576.116,Z 431.157,A -85,B 0,C 180,E1 27082.37,E2 27082.37} C_VEL
LIN {X 0,Y 576.095,Z 431.034,A -85,B 0,C 180,E1 27078.994,E2 27078.994} C_VEL
LIN {X 0,Y 576.122,Z 431.032,A -85,B 0,C 180,E1 27075.966,E2 27075.966} C_VEL
LIN {X 0,Y 576.083,Z 431.033,A -85,B 0,C 180,E1 27072.735,E2 27072.735} C_VEL
LIN {X 0,Y 576.138,Z 431.031,A -85,B 0,C 180,E1 27069.69,E2 27069.69} C_VEL
LIN {X 0,Y 576.077,Z 431.027,A -85,B 0,C 180,E1 27066.58,E2 27066.58} C_VEL
LIN {X 0,Y 576.143,Z 431.033,A -85,B 0,C 180,E1 27063.512,E2 27063.512} C_VEL
LIN {X 0,Y 576.072,Z 431.034,A -85,B 0,C 180,E1 27060.408,E2 27060.408} C_VEL
LIN {X 0,Y 576.148,Z 431.032,A -85,B 0,C 180,E1 27057.319,E2 27057.319} C_VEL
LIN {X 0,Y 576.074,Z 431.033,A -85,B 0,C 180,E1 27054.15,E2 27054.15} C_VEL
LIN {X 0,Y 576.142,Z 431.033,A -85,B 0,C 180,E1 27051.031,E2 27051.031} C_VEL
LIN {X 0,Y 576.08,Z 431.03,A -85,B 0,C 180,E1 27047.975,E2 27047.975} C_VEL
LIN {X 0,Y 576.129,Z 431.031,A -85,B 0,C 180,E1 27044.78,E2 27044.78} C_VEL
LIN {X 0,Y 576.09,Z 431.03,A -85,B 0,C 180,E1 27041.728,E2 27041.728} C_VEL
LIN {X 0,Y 576.105,Z 431.031,A -85,B 0,C 180,E1 27038.413,E2 27038.413} C_VEL
LIN {X 0,Y 576.106,Z 431.031,A -85,B 0,C 180,E1 27035.428,E2 27035.428} C_VEL
LIN {X 0,Y 576.095,Z 431.03,A -85,B 0,C 180,E1 27032.079,E2 27032.079} C_VEL
LIN {X 0,Y 576.137,Z 431.033,A -85,B 0,C 180,E1 27029.074,E2 27029.074} C_VEL
LIN {X 0,Y 576.095,Z 431.025,A -85,B 0,C 180,E1 27025.826,E2 27025.826} C_VEL
LIN {X 0,Y 576.162,Z 431.03,A -85,B 0,C 180,E1 27022.66,E2 27022.66} C_VEL
LIN {X 0,Y 576.099,Z 431.029,A -85,B 0,C 180,E1 27019.465,E2 27019.465} C_VEL
LIN {X 0,Y 576.143,Z 431.025,A -85,B 0,C 180,E1 27016.225,E2 27016.225} C_VEL
LIN {X 0,Y 576.113,Z 431.031,A -85,B 0,C 180,E1 27013.142,E2 27013.142} C_VEL
LIN {X 0,Y 576.116,Z 431.024,A -85,B 0,C 180,E1 27009.793,E2 27009.793} C_VEL
LIN {X 0,Y 576.148,Z 431.029,A -85,B 0,C 180,E1 27006.677,E2 27006.677} C_VEL
LIN {X 0,Y 576.111,Z 431.028,A -85,B 0,C 180,E1 27003.483,E2 27003.483} C_VEL
LIN {X 0,Y 576.158,Z 431.026,A -85,B 0,C 180,E1 27000.298,E2 27000.298} C_VEL
LIN {X 0,Y 576.113,Z 431.029,A -85,B 0,C 180,E1 26997.115,E2 26997.115} C_VEL
LIN {X 0,Y 576.153,Z 431.023,A -85,B 0,C 180,E1 26993.823,E2 26993.823} C_VEL
LIN {X 0,Y 576.136,Z 431.028,A -85,B 0,C 180,E1 26990.611,E2 26990.611} C_VEL
LIN {X 0,Y 576.123,Z 431.027,A -85,B 0,C 180,E1 26987.253,E2 26987.253} C_VEL
LIN {X 0,Y 576.157,Z 431.028,A -85,B 0,C 180,E1 26984.031,E2 26984.031} C_VEL
LIN {X 0,Y 576.124,Z 431.029,A -85,B 0,C 180,E1 26980.754,E2 26980.754} C_VEL
LIN {X 0,Y 576.155,Z 431.023,A -85,B 0,C 180,E1 26977.448,E2 26977.448} C_VEL
LIN {X 0,Y 576.154,Z 431.033,A -85,B 0,C 180,E1 26974.178,E2 26974.178} C_VEL
LIN {X 0,Y 576.13,Z 431.026,A -85,B 0,C 180,E1 26970.927,E2 26970.927} C_VEL
LIN {X 0,Y 576.152,Z 431.028,A -85,B 0,C 180,E1 26967.688,E2 26967.688} C_VEL
LIN {X 0,Y 576.132,Z 431.029,A -85,B 0,C 180,E1 26964.452,E2 26964.452} C_VEL
LIN {X 0,Y 576.157,Z 431.023,A -85,B 0,C 180,E1 26961.187,E2 26961.187} C_VEL
LIN {X 0,Y 576.154,Z 431.031,A -85,B 0,C 180,E1 26957.809,E2 26957.809} C_VEL
LIN {X 0,Y 576.136,Z 431.026,A -85,B 0,C 180,E1 26954.498,E2 26954.498} C_VEL
LIN {X 0,Y 576.148,Z 431.027,A -85,B 0,C 180,E1 26951.259,E2 26951.259} C_VEL
LIN {X 0,Y 576.145,Z 431.032,A -85,B 0,C 180,E1 26948.012,E2 26948.012} C_VEL
LIN {X 0,Y 576.152,Z 431.025,A -85,B 0,C 180,E1 26944.656,E2 26944.656} C_VEL
LIN {X 0,Y 576.155,Z 431.107,A -85,B 0,C 180,E1 26941.357,E2 26941.357} C_VEL
LIN {X 0,Y 576.325,Z 432.001,A -85,B 0,C 180,E1 26941.207,E2 26941.207} C_VEL
LIN {X 0,Y 578.905,Z 439.399,A -85,B 0,C 180,E1 26940.517,E2 26940.517} C_VEL
LIN {X 0,Y 578.319,Z 484.373,A -85,B 0,C 180,E1 26937.319,E2 26937.319} C_VEL
LIN {X 0,Y 577.785,Z 529.978,A -85,B 0,C 180,E1 26934.159,E2 26934.159} C_VEL
LIN {X 0,Y 577.805,Z 539.211,A -85,B 0,C 180,E1 26933.558,E2 26933.558} C_VEL
LIN {X 0,Y 578.387,Z 545.267,A -85,B 0,C 180,E1 26933.449,E2 26933.449} C_VEL
LIN {X 0,Y 577.839,Z 748.31,A -85,B 0,C 180,E1 26930.777,E2 26930.777} C_VEL
LIN {X 0,Y 577.664,Z 767.343,A -85,B 0,C 180,E1 26930.336,E2 26930.336} C_VEL
LIN {X 0,Y 577.483,Z 785.398,A -85,B 0,C 180,E1 26929.732,E2 26929.732} C_VEL
LIN {X 0,Y 577.257,Z 803.378,A -85,B 0,C 180,E1 26928.934,E2 26928.934} C_VEL
LIN {X 0,Y 577.027,Z 820.588,A -85,B 0,C 180,E1 26927.965,E2 26927.965} C_VEL
LIN {X 0,Y 576.798,Z 836.182,A -85,B 0,C 180,E1 26926.889,E2 26926.889} C_VEL
LIN {X 0,Y 576.571,Z 851.113,A -85,B 0,C 180,E1 26925.644,E2 26925.644} C_VEL
LIN {X 0,Y 576.369,Z 864.944,A -85,B 0,C 180,E1 26924.261,E2 26924.261} C_VEL
LIN {X 0,Y 576.208,Z 877.684,A -85,B 0,C 180,E1 26922.731,E2 26922.731} C_VEL
LIN {X 0,Y 576.085,Z 888.866,A -85,B 0,C 180,E1 26921.108,E2 26921.108} C_VEL
LIN {X 0,Y 575.999,Z 898.509,A -85,B 0,C 180,E1 26919.391,E2 26919.391} C_VEL
LIN {X 0,Y 575.955,Z 906.177,A -85,B 0,C 180,E1 26917.682,E2 26917.682} C_VEL
LIN {X 0,Y 575.921,Z 912.491,A -85,B 0,C 180,E1 26915.853,E2 26915.853} C_VEL
LIN {X 0,Y 575.92,Z 916.875,A -85,B 0,C 180,E1 26914.082,E2 26914.082} C_VEL
LIN {X 0,Y 575.916,Z 919.79,A -85,B 0,C 180,E1 26912.189,E2 26912.189} C_VEL
LIN {X 0,Y 575.907,Z 920.94,A -85,B 0,C 180,E1 26910.299,E2 26910.299} C_VEL
LIN {X 0,Y 575.914,Z 920.349,A -85,B 0,C 180,E1 26908.408,E2 26908.408} C_VEL
LIN {X 0,Y 575.908,Z 918.005,A -85,B 0,C 180,E1 26906.516,E2 26906.516} C_VEL
LIN {X 0,Y 575.919,Z 914.098,A -85,B 0,C 180,E1 26904.721,E2 26904.721} C_VEL
LIN {X 0,Y 575.94,Z 908.469,A -85,B 0,C 180,E1 26902.92,E2 26902.92} C_VEL
LIN {X 0,Y 575.976,Z 901.425,A -85,B 0,C 180,E1 26901.213,E2 26901.213} C_VEL
LIN {X 0,Y 576.053,Z 892.513,A -85,B 0,C 180,E1 26899.499,E2 26899.499} C_VEL
LIN {X 0,Y 576.156,Z 882.149,A -85,B 0,C 180,E1 26897.879,E2 26897.879} C_VEL
LIN {X 0,Y 576.308,Z 869.945,A -85,B 0,C 180,E1 26896.304,E2 26896.304} C_VEL
LIN {X 0,Y 576.496,Z 856.579,A -85,B 0,C 180,E1 26894.869,E2 26894.869} C_VEL
LIN {X 0,Y 576.718,Z 841.601,A -85,B 0,C 180,E1 26893.533,E2 26893.533} C_VEL
LIN {X 0,Y 576.96,Z 825.427,A -85,B 0,C 180,E1 26892.346,E2 26892.346} C_VEL
LIN {X 0,Y 577.171,Z 809.191,A -85,B 0,C 180,E1 26891.368,E2 26891.368} C_VEL
LIN {X 0,Y 577.424,Z 791.802,A -85,B 0,C 180,E1 26890.529,E2 26890.529} C_VEL
LIN {X 0,Y 577.605,Z 773.741,A -85,B 0,C 180,E1 26889.857,E2 26889.857} C_VEL
LIN {X 0,Y 577.785,Z 755.309,A -85,B 0,C 180,E1 26889.364,E2 26889.364} C_VEL
LIN {X 0,Y 577.901,Z 735.364,A -85,B 0,C 180,E1 26889.03,E2 26889.03} C_VEL
LIN {X 0,Y 578.222,Z 541.866,A -85,B 0,C 180,E1 26886.499,E2 26886.499} C_VEL
LIN {X 0,Y 577.719,Z 537.884,A -85,B 0,C 180,E1 26886.381,E2 26886.381} C_VEL
LIN {X 0,Y 578.234,Z 491.389,A -85,B 0,C 180,E1 26883.172,E2 26883.172} C_VEL
LIN {X 0,Y 578.81,Z 446.494,A -85,B 0,C 180,E1 26879.994,E2 26879.994} C_VEL
LIN {X 0,Y 578.83,Z 438.999,A -85,B 0,C 180,E1 26879.45,E2 26879.45} C_VEL
LIN {X 0,Y 576.192,Z 431.354,A -85,B 0,C 180,E1 26878.716,E2 26878.716} C_VEL
LIN {X 0,Y 576.141,Z 431.027,A -85,B 0,C 180,E1 26877.876,E2 26877.876} C_VEL
LIN {X 0,Y 576.146,Z 431.032,A -85,B 0,C 180,E1 26874.576,E2 26874.576} C_VEL
LIN {X 0,Y 576.156,Z 431.023,A -85,B 0,C 180,E1 26871.209,E2 26871.209} C_VEL
LIN {X 0,Y 576.151,Z 431.031,A -85,B 0,C 180,E1 26867.943,E2 26867.943} C_VEL
LIN {X 0,Y 576.146,Z 431.026,A -85,B 0,C 180,E1 26864.641,E2 26864.641} C_VEL
LIN {X 0,Y 576.14,Z 431.027,A -85,B 0,C 180,E1 26861.392,E2 26861.392} C_VEL
LIN {X 0,Y 576.15,Z 431.029,A -85,B 0,C 180,E1 26858.156,E2 26858.156} C_VEL
LIN {X 0,Y 576.154,Z 431.023,A -85,B 0,C 180,E1 26854.816,E2 26854.816} C_VEL
LIN {X 0,Y 576.143,Z 431.03,A -85,B 0,C 180,E1 26851.491,E2 26851.491} C_VEL
LIN {X 0,Y 576.147,Z 431.025,A -85,B 0,C 180,E1 26848.279,E2 26848.279} C_VEL
LIN {X 0,Y 576.137,Z 431.026,A -85,B 0,C 180,E1 26845.052,E2 26845.052} C_VEL
LIN {X 0,Y 576.149,Z 431.03,A -85,B 0,C 180,E1 26841.801,E2 26841.801} C_VEL
LIN {X 0,Y 576.155,Z 431.022,A -85,B 0,C 180,E1 26838.516,E2 26838.516} C_VEL
LIN {X 0,Y 576.143,Z 431.027,A -85,B 0,C 180,E1 26835.192,E2 26835.192} C_VEL
LIN {X 0,Y 576.147,Z 431.026,A -85,B 0,C 180,E1 26831.918,E2 26831.918} C_VEL
LIN {X 0,Y 576.135,Z 431.026,A -85,B 0,C 180,E1 26828.684,E2 26828.684} C_VEL
LIN {X 0,Y 576.151,Z 431.03,A -85,B 0,C 180,E1 26825.477,E2 26825.477} C_VEL
LIN {X 0,Y 576.15,Z 431.024,A -85,B 0,C 180,E1 26822.188,E2 26822.188} C_VEL
LIN {X 0,Y 576.141,Z 431.03,A -85,B 0,C 180,E1 26818.807,E2 26818.807} C_VEL
LIN {X 0,Y 576.149,Z 431.026,A -85,B 0,C 180,E1 26815.521,E2 26815.521} C_VEL
LIN {X 0,Y 576.134,Z 431.026,A -85,B 0,C 180,E1 26812.284,E2 26812.284} C_VEL
LIN {X 0,Y 576.157,Z 431.03,A -85,B 0,C 180,E1 26808.995,E2 26808.995} C_VEL
LIN {X 0,Y 576.156,Z 431.021,A -85,B 0,C 180,E1 26805.631,E2 26805.631} C_VEL
LIN {X 0,Y 576.151,Z 431.027,A -85,B 0,C 180,E1 26803.306,E2 26803.306} C_VEL
LIN {X 0,Y 575.151,Z 431.157,A -85,B 0,C 180,E1 26802.54,E2 26802.54} C_VEL
LIN {X 0,Y 568.709,Z 431.957,A -85,B 0,C 180,E1 26800.39,E2 26800.39} C_VEL
LIN {X 0,Y 568.203,Z 432.014,A -85,B 0,C 180,E1 26799.83,E2 26799.83} C_VEL
LIN {X 0,Y 568.206,Z 432.019,A -85,B 0,C 180,E1 26796.456,E2 26796.456} C_VEL
LIN {X 0,Y 568.214,Z 432.015,A -85,B 0,C 180,E1 26793.144,E2 26793.144} C_VEL
LIN {X 0,Y 568.193,Z 432.017,A -85,B 0,C 180,E1 26789.899,E2 26789.899} C_VEL
LIN {X 0,Y 568.218,Z 432.021,A -85,B 0,C 180,E1 26786.58,E2 26786.58} C_VEL
LIN {X 0,Y 568.218,Z 432.014,A -85,B 0,C 180,E1 26783.191,E2 26783.191} C_VEL
LIN {X 0,Y 568.194,Z 432.022,A -85,B 0,C 180,E1 26779.905,E2 26779.905} C_VEL
LIN {X 0,Y 568.219,Z 432.202,A -85,B 0,C 180,E1 26777.868,E2 26777.868} C_VEL
LIN {X 0,Y 570.052,Z 439.926,A -85,B 0,C 180,E1 26776.838,E2 26776.838} C_VEL
LIN {X 0,Y 569.449,Z 468.906,A -85,B 0,C 180,E1 26773.495,E2 26773.495} C_VEL
LIN {X 0,Y 569.063,Z 498.477,A -85,B 0,C 180,E1 26770.218,E2 26770.218} C_VEL
LIN {X 0,Y 568.719,Z 529.265,A -85,B 0,C 180,E1 26766.876,E2 26766.876} C_VEL
LIN {X 0,Y 568.458,Z 556.924,A -85,B 0,C 180,E1 26763.949,E2 26763.949} C_VEL
LIN {X 0,Y 568.991,Z 563.684,A -85,B 0,C 180,E1 26763.834,E2 26763.834} C_VEL
LIN {X 0,Y 568.747,Z 668.444,A -85,B 0,C 180,E1 26762.482,E2 26762.482} C_VEL
LIN {X 0,Y 568.685,Z 683.356,A -85,B 0,C 180,E1 26762.101,E2 26762.101} C_VEL
LIN {X 0,Y 568.563,Z 697.427,A -85,B 0,C 180,E1 26761.545,E2 26761.545} C_VEL
LIN {X 0,Y 568.412,Z 710.168,A -85,B 0,C 180,E1 26760.861,E2 26760.861} C_VEL
LIN {X 0,Y 568.274,Z 722.728,A -85,B 0,C 180,E1 26759.979,E2 26759.979} C_VEL
LIN {X 0,Y 568.163,Z 734.186,A -85,B 0,C 180,E1 26758.943,E2 26758.943} C_VEL
LIN {X 0,Y 568.064,Z 744.137,A -85,B 0,C 180,E1 26757.803,E2 26757.803} C_VEL
LIN {X 0,Y 567.993,Z 752.654,A -85,B 0,C 180,E1 26756.559,E2 26756.559} C_VEL
LIN {X 0,Y 567.946,Z 759.77,A -85,B 0,C 180,E1 26755.191,E2 26755.191} C_VEL
LIN {X 0,Y 567.926,Z 765.141,A -85,B 0,C 180,E1 26753.776,E2 26753.776} C_VEL
LIN {X 0,Y 567.918,Z 768.936,A -85,B 0,C 180,E1 26752.242,E2 26752.242} C_VEL
LIN {X 0,Y 567.916,Z 770.745,A -85,B 0,C 180,E1 26750.724,E2 26750.724} C_VEL
LIN {X 0,Y 567.916,Z 770.769,A -85,B 0,C 180,E1 26749.222,E2 26749.222} C_VEL
LIN {X 0,Y 567.917,Z 769.05,A -85,B 0,C 180,E1 26747.733,E2 26747.733} C_VEL
LIN {X 0,Y 567.925,Z 765.506,A -85,B 0,C 180,E1 26746.256,E2 26746.256} C_VEL
LIN {X 0,Y 567.943,Z 760.449,A -85,B 0,C 180,E1 26744.869,E2 26744.869} C_VEL
LIN {X 0,Y 567.989,Z 753.16,A -85,B 0,C 180,E1 26743.436,E2 26743.436} C_VEL
LIN {X 0,Y 568.057,Z 744.791,A -85,B 0,C 180,E1 26742.193,E2 26742.193} C_VEL
LIN {X 0,Y 568.154,Z 735.103,A -85,B 0,C 180,E1 26741.059,E2 26741.059} C_VEL
LIN {X 0,Y 568.284,Z 723.342,A -85,B 0,C 180,E1 26739.98,E2 26739.98} C_VEL
LIN {X 0,Y 568.417,Z 710.297,A -85,B 0,C 180,E1 26739.058,E2 26739.058} C_VEL
LIN {X 0,Y 568.566,Z 696.931,A -85,B 0,C 180,E1 26738.342,E2 26738.342} C_VEL
LIN {X 0,Y 568.699,Z 682.436,A -85,B 0,C 180,E1 26737.78,E2 26737.78} C_VEL
LIN {X 0,Y 568.79,Z 666.719,A -85,B 0,C 180,E1 26737.395,E2 26737.395} C_VEL
LIN {X 0,Y 568.777,Z 559.197,A -85,B 0,C 180,E1 26736.013,E2 26736.013} C_VEL
LIN {X 0,Y 568.489,Z 556.797,A -85,B 0,C 180,E1 26735.956,E2 26735.956} C_VEL
LIN {X 0,Y 568.717,Z 526.364,A -85,B 0,C 180,E1 26732.721,E2 26732.721} C_VEL
LIN {X 0,Y 569.098,Z 495.78,A -85,B 0,C 180,E1 26729.396,E2 26729.396} C_VEL
LIN {X 0,Y 569.493,Z 465.877,A -85,B 0,C 180,E1 26726.074,E2 26726.074} C_VEL
LIN {X 0,Y 569.964,Z 439.069,A -85,B 0,C 180,E1 26722.997,E2 26722.997} C_VEL
LIN {X 0,Y 568.204,Z 432.117,A -85,B 0,C 180,E1 26722.034,E2 26722.034} C_VEL
LIN {X 0,Y 568.149,Z 432.024,A -85,B 0,C 180,E1 26718.838,E2 26718.838} C_VEL
LIN {X 0,Y 568.211,Z 432.021,A -85,B 0,C 180,E1 26715.738,E2 26715.738} C_VEL
LIN {X 0,Y 568.141,Z 432.022,A -85,B 0,C 180,E1 26712.591,E2 26712.591} C_VEL
LIN {X 0,Y 568.21,Z 432.023,A -85,B 0,C 180,E1 26709.414,E2 26709.414} C_VEL
LIN {X 0,Y 568.137,Z 432.014,A -85,B 0,C 180,E1 26706.343,E2 26706.343} C_VEL
LIN {X 0,Y 568.182,Z 432.022,A -85,B 0,C 180,E1 26703.111,E2 26703.111} C_VEL
LIN {X 0,Y 568.136,Z 432.023,A -85,B 0,C 180,E1 26700.129,E2 26700.129} C_VEL
LIN {X 0,Y 568.167,Z 432.022,A -85,B 0,C 180,E1 26696.895,E2 26696.895} C_VEL
LIN {X 0,Y 568.146,Z 432.021,A -85,B 0,C 180,E1 26693.874,E2 26693.874} C_VEL
LIN {X 0,Y 568.154,Z 432.022,A -85,B 0,C 180,E1 26690.557,E2 26690.557} C_VEL
LIN {X 0,Y 568.16,Z 432.019,A -85,B 0,C 180,E1 26687.622,E2 26687.622} C_VEL
LIN {X 0,Y 568.149,Z 432.021,A -85,B 0,C 180,E1 26684.32,E2 26684.32} C_VEL
LIN {X 0,Y 568.188,Z 432.019,A -85,B 0,C 180,E1 26681.287,E2 26681.287} C_VEL
LIN {X 0,Y 568.151,Z 432.02,A -85,B 0,C 180,E1 26678.126,E2 26678.126} C_VEL
LIN {X 0,Y 568.214,Z 432.017,A -85,B 0,C 180,E1 26675.005,E2 26675.005} C_VEL
LIN {X 0,Y 568.152,Z 432.019,A -85,B 0,C 180,E1 26671.787,E2 26671.787} C_VEL
LIN {X 0,Y 568.216,Z 432.015,A -85,B 0,C 180,E1 26668.59,E2 26668.59} C_VEL
LIN {X 0,Y 568.162,Z 432.014,A -85,B 0,C 180,E1 26665.429,E2 26665.429} C_VEL
LIN {X 0,Y 568.17,Z 432.018,A -85,B 0,C 180,E1 26662.014,E2 26662.014} C_VEL
LIN {X 0,Y 568.204,Z 432.02,A -85,B 0,C 180,E1 26658.892,E2 26658.892} C_VEL
LIN {X 0,Y 568.163,Z 432.016,A -85,B 0,C 180,E1 26655.62,E2 26655.62} C_VEL
LIN {X 0,Y 568.223,Z 432.016,A -85,B 0,C 180,E1 26652.397,E2 26652.397} C_VEL
LIN {X 0,Y 568.171,Z 432.015,A -85,B 0,C 180,E1 26649.162,E2 26649.162} C_VEL
LIN {X 0,Y 568.193,Z 432.015,A -85,B 0,C 180,E1 26645.858,E2 26645.858} C_VEL
LIN {X 0,Y 568.209,Z 432.021,A -85,B 0,C 180,E1 26642.622,E2 26642.622} C_VEL
LIN {X 0,Y 568.174,Z 432.012,A -85,B 0,C 180,E1 26639.395,E2 26639.395} C_VEL
LIN {X 0,Y 568.222,Z 432.017,A -85,B 0,C 180,E1 26636.125,E2 26636.125} C_VEL
LIN {X 0,Y 568.179,Z 432.016,A -85,B 0,C 180,E1 26632.924,E2 26632.924} C_VEL
LIN {X 0,Y 568.199,Z 432.014,A -85,B 0,C 180,E1 26629.558,E2 26629.558} C_VEL
LIN {X 0,Y 568.219,Z 432.018,A -85,B 0,C 180,E1 26626.246,E2 26626.246} C_VEL
LIN {X 0,Y 568.182,Z 432.015,A -85,B 0,C 180,E1 26623.015,E2 26623.015} C_VEL
LIN {X 0,Y 568.219,Z 432.012,A -85,B 0,C 180,E1 26619.718,E2 26619.718} C_VEL
LIN {X 0,Y 568.197,Z 432.019,A -85,B 0,C 180,E1 26616.456,E2 26616.456} C_VEL
LIN {X 0,Y 568.198,Z 432.011,A -85,B 0,C 180,E1 26613.112,E2 26613.112} C_VEL
LIN {X 0,Y 568.219,Z 432.018,A -85,B 0,C 180,E1 26609.901,E2 26609.901} C_VEL
LIN {X 0,Y 568.192,Z 432.016,A -85,B 0,C 180,E1 26606.699,E2 26606.699} C_VEL
LIN {X 0,Y 568.217,Z 432.014,A -85,B 0,C 180,E1 26603.36,E2 26603.36} C_VEL
LIN {X 0,Y 568.221,Z 432.019,A -85,B 0,C 180,E1 26599.946,E2 26599.946} C_VEL
LIN {X 0,Y 568.198,Z 432.015,A -85,B 0,C 180,E1 26596.615,E2 26596.615} C_VEL
LIN {X 0,Y 568.21,Z 432.017,A -85,B 0,C 180,E1 26593.336,E2 26593.336} C_VEL
LIN {X 0,Y 568.205,Z 432.021,A -85,B 0,C 180,E1 26590.052,E2 26590.052} C_VEL
LIN {X 0,Y 568.21,Z 432.015,A -85,B 0,C 180,E1 26586.622,E2 26586.622} C_VEL
LIN {X 0,Y 568.206,Z 432.016,A -85,B 0,C 180,E1 26583.296,E2 26583.296} C_VEL
LIN {X 0,Y 568.246,Z 432.22,A -85,B 0,C 180,E1 26581.684,E2 26581.684} C_VEL
LIN {X 0,Y 570.955,Z 440.181,A -85,B 0,C 180,E1 26580.897,E2 26580.897} C_VEL
LIN {X 0,Y 571.591,Z 443.053,A -85,B 0,C 180,E1 26580.658,E2 26580.658} C_VEL
LIN {X 0,Y 570.94,Z 486.658,A -85,B 0,C 180,E1 26577.538,E2 26577.538} C_VEL
LIN {X 0,Y 570.271,Z 532.341,A -85,B 0,C 180,E1 26574.332,E2 26574.332} C_VEL
LIN {X 0,Y 570.302,Z 539.288,A -85,B 0,C 180,E1 26573.885,E2 26573.885} C_VEL
LIN {X 0,Y 571.044,Z 546.03,A -85,B 0,C 180,E1 26573.758,E2 26573.758} C_VEL
LIN {X 0,Y 570.357,Z 748.31,A -85,B 0,C 180,E1 26571.062,E2 26571.062} C_VEL
LIN {X 0,Y 570.145,Z 767.342,A -85,B 0,C 180,E1 26570.617,E2 26570.617} C_VEL
LIN {X 0,Y 569.912,Z 785.397,A -85,B 0,C 180,E1 26570.006,E2 26570.006} C_VEL
LIN {X 0,Y 569.635,Z 803.18,A -85,B 0,C 180,E1 26569.208,E2 26569.208} C_VEL
LIN {X 0,Y 569.348,Z 819.774,A -85,B 0,C 180,E1 26568.269,E2 26568.269} C_VEL
LIN {X 0,Y 569.055,Z 835.629,A -85,B 0,C 180,E1 26567.169,E2 26567.169} C_VEL
LIN {X 0,Y 568.769,Z 850.557,A -85,B 0,C 180,E1 26565.917,E2 26565.917} C_VEL
LIN {X 0,Y 568.524,Z 864.018,A -85,B 0,C 180,E1 26564.566,E2 26564.566} C_VEL
LIN {X 0,Y 568.307,Z 876.911,A -85,B 0,C 180,E1 26563.015,E2 26563.015} C_VEL
LIN {X 0,Y 568.142,Z 888.228,A -85,B 0,C 180,E1 26561.368,E2 26561.368} C_VEL
LIN {X 0,Y 568.032,Z 897.993,A -85,B 0,C 180,E1 26559.626,E2 26559.626} C_VEL
LIN {X 0,Y 567.966,Z 905.772,A -85,B 0,C 180,E1 26557.893,E2 26557.893} C_VEL
LIN {X 0,Y 567.932,Z 912.109,A -85,B 0,C 180,E1 26556.064,E2 26556.064} C_VEL
LIN {X 0,Y 567.919,Z 916.875,A -85,B 0,C 180,E1 26554.14,E2 26554.14} C_VEL
LIN {X 0,Y 567.916,Z 919.79,A -85,B 0,C 180,E1 26552.22,E2 26552.22} C_VEL
LIN {X 0,Y 567.907,Z 920.94,A -85,B 0,C 180,E1 26550.303,E2 26550.303} C_VEL
LIN {X 0,Y 567.914,Z 920.348,A -85,B 0,C 180,E1 26548.386,E2 26548.386} C_VEL
LIN {X 0,Y 567.909,Z 918.005,A -85,B 0,C 180,E1 26546.467,E2 26546.467} C_VEL
LIN {X 0,Y 567.923,Z 914.098,A -85,B 0,C 180,E1 26544.646,E2 26544.646} C_VEL
LIN {X 0,Y 567.947,Z 908.469,A -85,B 0,C 180,E1 26542.82,E2 26542.82} C_VEL
LIN {X 0,Y 568,Z 901.426,A -85,B 0,C 180,E1 26541.089,E2 26541.089} C_VEL
LIN {X 0,Y 568.093,Z 892.514,A -85,B 0,C 180,E1 26539.351,E2 26539.351} C_VEL
LIN {X 0,Y 568.23,Z 882.151,A -85,B 0,C 180,E1 26537.707,E2 26537.707} C_VEL
LIN {X 0,Y 568.414,Z 870.35,A -85,B 0,C 180,E1 26536.159,E2 26536.159} C_VEL
LIN {X 0,Y 568.647,Z 857.085,A -85,B 0,C 180,E1 26534.708,E2 26534.708} C_VEL
LIN {X 0,Y 568.927,Z 842.228,A -85,B 0,C 180,E1 26533.354,E2 26533.354} C_VEL
LIN {X 0,Y 569.235,Z 826.232,A -85,B 0,C 180,E1 26532.151,E2 26532.151} C_VEL
LIN {X 0,Y 569.518,Z 809.145,A -85,B 0,C 180,E1 26531.106,E2 26531.106} C_VEL
LIN {X 0,Y 569.828,Z 791.805,A -85,B 0,C 180,E1 26530.259,E2 26530.259} C_VEL
LIN {X 0,Y 570.066,Z 773.636,A -85,B 0,C 180,E1 26529.575,E2 26529.575} C_VEL
LIN {X 0,Y 570.29,Z 755.147,A -85,B 0,C 180,E1 26529.077,E2 26529.077} C_VEL
LIN {X 0,Y 570.432,Z 735.07,A -85,B 0,C 180,E1 26528.739,E2 26528.739} C_VEL
LIN {X 0,Y 570.879,Z 542.938,A -85,B 0,C 180,E1 26526.193,E2 26526.193} C_VEL
LIN {X 0,Y 570.216,Z 538.331,A -85,B 0,C 180,E1 26526.078,E2 26526.078} C_VEL
LIN {X 0,Y 570.846,Z 492.964,A -85,B 0,C 180,E1 26522.909,E2 26522.909} C_VEL
LIN {X 0,Y 571.542,Z 447.933,A -85,B 0,C 180,E1 26519.689,E2 26519.689} C_VEL
LIN {X 0,Y 571.409,Z 441.513,A -85,B 0,C 180,E1 26519.222,E2 26519.222} C_VEL
LIN {X 0,Y 568.271,Z 432.374,A -85,B 0,C 180,E1 26518.351,E2 26518.351} C_VEL
LIN {X 0,Y 568.202,Z 432.015,A -85,B 0,C 180,E1 26517.779,E2 26517.779} C_VEL
LIN {X 0,Y 568.21,Z 432.021,A -85,B 0,C 180,E1 26514.501,E2 26514.501} C_VEL
LIN {X 0,Y 568.217,Z 432.012,A -85,B 0,C 180,E1 26511.083,E2 26511.083} C_VEL
LIN {X 0,Y 568.204,Z 432.018,A -85,B 0,C 180,E1 26507.763,E2 26507.763} C_VEL
LIN {X 0,Y 568.206,Z 432.016,A -85,B 0,C 180,E1 26504.548,E2 26504.548} C_VEL
LIN {X 0,Y 568.203,Z 432.015,A -85,B 0,C 180,E1 26501.29,E2 26501.29} C_VEL
LIN {X 0,Y 568.219,Z 432.022,A -85,B 0,C 180,E1 26497.887,E2 26497.887} C_VEL
LIN {X 0,Y 568.212,Z 432.014,A -85,B 0,C 180,E1 26494.514,E2 26494.514} C_VEL
LIN {X 0,Y 568.199,Z 432.016,A -85,B 0,C 180,E1 26491.217,E2 26491.217} C_VEL
LIN {X 0,Y 568.213,Z 432.017,A -85,B 0,C 180,E1 26487.951,E2 26487.951} C_VEL
LIN {X 0,Y 568.213,Z 432.011,A -85,B 0,C 180,E1 26484.648,E2 26484.648} C_VEL
LIN {X 0,Y 568.203,Z 432.018,A -85,B 0,C 180,E1 26481.253,E2 26481.253} C_VEL
LIN {X 0,Y 568.208,Z 432.015,A -85,B 0,C 180,E1 26477.935,E2 26477.935} C_VEL
LIN {X 0,Y 568.202,Z 432.01,A -85,B 0,C 180,E1 26474.678,E2 26474.678} C_VEL
LIN {X 0,Y 568.218,Z 432.021,A -85,B 0,C 180,E1 26471.366,E2 26471.366} C_VEL
LIN {X 0,Y 568.214,Z 432.012,A -85,B 0,C 180,E1 26467.991,E2 26467.991} C_VEL
LIN {X 0,Y 568.197,Z 432.014,A -85,B 0,C 180,E1 26464.744,E2 26464.744} C_VEL
LIN {X 0,Y 568.21,Z 432.018,A -85,B 0,C 180,E1 26461.512,E2 26461.512} C_VEL
LIN {X 0,Y 568.201,Z 432.014,A -85,B 0,C 180,E1 26458.286,E2 26458.286} C_VEL
LIN {X 0,Y 568.214,Z 432.018,A -85,B 0,C 180,E1 26454.952,E2 26454.952} C_VEL
LIN {X 0,Y 568.214,Z 432.014,A -85,B 0,C 180,E1 26451.602,E2 26451.602} C_VEL
LIN {X 0,Y 568.195,Z 432.017,A -85,B 0,C 180,E1 26448.324,E2 26448.324} C_VEL
LIN {X 0,Y 568.215,Z 432.018,A -85,B 0,C 180,E1 26445.009,E2 26445.009} C_VEL
LIN {X 0,Y 568.215,Z 432.011,A -85,B 0,C 180,E1 26441.64,E2 26441.64} C_VEL
LIN {X 0,Y 568.203,Z 432.014,A -85,B 0,C 180,E1 26439.83,E2 26439.83} C_VEL
LIN {X 0,Y 567.251,Z 432.138,A -85,B 0,C 180,E1 26439.053,E2 26439.053} C_VEL
LIN {X 0,Y 560.716,Z 432.956,A -85,B 0,C 180,E1 26436.816,E2 26436.816} C_VEL
LIN {X 0,Y 560.26,Z 433.006,A -85,B 0,C 180,E1 26436.304,E2 26436.304} C_VEL
LIN {X 0,Y 560.273,Z 433.006,A -85,B 0,C 180,E1 26433.045,E2 26433.045} C_VEL
LIN {X 0,Y 560.257,Z 433.005,A -85,B 0,C 180,E1 26429.742,E2 26429.742} C_VEL
LIN {X 0,Y 560.277,Z 433.01,A -85,B 0,C 180,E1 26426.411,E2 26426.411} C_VEL
LIN {X 0,Y 560.279,Z 433.005,A -85,B 0,C 180,E1 26423.029,E2 26423.029} C_VEL
LIN {X 0,Y 560.253,Z 433.01,A -85,B 0,C 180,E1 26419.756,E2 26419.756} C_VEL
LIN {X 0,Y 560.311,Z 433.269,A -85,B 0,C 180,E1 26418.196,E2 26418.196} C_VEL
LIN {X 0,Y 562.525,Z 442.542,A -85,B 0,C 180,E1 26416.957,E2 26416.957} C_VEL
LIN {X 0,Y 561.817,Z 471.411,A -85,B 0,C 180,E1 26413.586,E2 26413.586} C_VEL
LIN {X 0,Y 561.3,Z 500.168,A -85,B 0,C 180,E1 26410.322,E2 26410.322} C_VEL
LIN {X 0,Y 560.876,Z 531.051,A -85,B 0,C 180,E1 26406.924,E2 26406.924} C_VEL
LIN {X 0,Y 560.587,Z 556.988,A -85,B 0,C 180,E1 26404.148,E2 26404.148} C_VEL
LIN {X 0,Y 561.223,Z 564.197,A -85,B 0,C 180,E1 26404.024,E2 26404.024} C_VEL
LIN {X 0,Y 560.935,Z 668.49,A -85,B 0,C 180,E1 26402.658,E2 26402.658} C_VEL
LIN {X 0,Y 560.857,Z 683.044,A -85,B 0,C 180,E1 26402.284,E2 26402.284} C_VEL
LIN {X 0,Y 560.703,Z 697.774,A -85,B 0,C 180,E1 26401.694,E2 26401.694} C_VEL
LIN {X 0,Y 560.517,Z 710.845,A -85,B 0,C 180,E1 26400.973,E2 26400.973} C_VEL
LIN {X 0,Y 560.351,Z 723.375,A -85,B 0,C 180,E1 26400.07,E2 26400.07} C_VEL
LIN {X 0,Y 560.204,Z 735.606,A -85,B 0,C 180,E1 26398.926,E2 26398.926} C_VEL
LIN {X 0,Y 560.077,Z 746.077,A -85,B 0,C 180,E1 26397.655,E2 26397.655} C_VEL
LIN {X 0,Y 559.997,Z 754.114,A -85,B 0,C 180,E1 26396.396,E2 26396.396} C_VEL
LIN {X 0,Y 559.95,Z 760.785,A -85,B 0,C 180,E1 26395.036,E2 26395.036} C_VEL
LIN {X 0,Y 559.925,Z 766.215,A -85,B 0,C 180,E1 26393.466,E2 26393.466} C_VEL
LIN {X 0,Y 559.919,Z 769.338,A -85,B 0,C 180,E1 26392.024,E2 26392.024} C_VEL
LIN {X 0,Y 559.917,Z 770.888,A -85,B 0,C 180,E1 26390.487,E2 26390.487} C_VEL
LIN {X 0,Y 559.916,Z 770.521,A -85,B 0,C 180,E1 26388.837,E2 26388.837} C_VEL
LIN {X 0,Y 559.918,Z 768.153,A -85,B 0,C 180,E1 26387.243,E2 26387.243} C_VEL
LIN {X 0,Y 559.93,Z 764.43,A -85,B 0,C 180,E1 26385.855,E2 26385.855} C_VEL
LIN {X 0,Y 559.963,Z 758.547,A -85,B 0,C 180,E1 26384.371,E2 26384.371} C_VEL
LIN {X 0,Y 560.024,Z 751.074,A -85,B 0,C 180,E1 26383,E2 26383} C_VEL
LIN {X 0,Y 560.121,Z 742.156,A -85,B 0,C 180,E1 26381.741,E2 26381.741} C_VEL
LIN {X 0,Y 560.255,Z 731.768,A -85,B 0,C 180,E1 26380.592,E2 26380.592} C_VEL
LIN {X 0,Y 560.411,Z 719.687,A -85,B 0,C 180,E1 26379.551,E2 26379.551} C_VEL
LIN {X 0,Y 560.578,Z 707.278,A -85,B 0,C 180,E1 26378.72,E2 26378.72} C_VEL
LIN {X 0,Y 560.75,Z 694.075,A -85,B 0,C 180,E1 26378.046,E2 26378.046} C_VEL
LIN {X 0,Y 560.89,Z 679.16,A -85,B 0,C 180,E1 26377.509,E2 26377.509} C_VEL
LIN {X 0,Y 560.99,Z 664.469,A -85,B 0,C 180,E1 26377.181,E2 26377.181} C_VEL
LIN {X 0,Y 560.997,Z 559.868,A -85,B 0,C 180,E1 26375.825,E2 26375.825} C_VEL
LIN {X 0,Y 560.613,Z 556.519,A -85,B 0,C 180,E1 26375.732,E2 26375.732} C_VEL
LIN {X 0,Y 560.899,Z 526.174,A -85,B 0,C 180,E1 26372.452,E2 26372.452} C_VEL
LIN {X 0,Y 561.357,Z 495.62,A -85,B 0,C 180,E1 26369.081,E2 26369.081} C_VEL
LIN {X 0,Y 561.877,Z 466.849,A -85,B 0,C 180,E1 26365.816,E2 26365.816} C_VEL
LIN {X 0,Y 562.38,Z 441.376,A -85,B 0,C 180,E1 26362.851,E2 26362.851} C_VEL
LIN {X 0,Y 560.291,Z 433.08,A -85,B 0,C 180,E1 26361.689,E2 26361.689} C_VEL
LIN {X 0,Y 560.211,Z 433.012,A -85,B 0,C 180,E1 26358.48,E2 26358.48} C_VEL
LIN {X 0,Y 560.239,Z 433.012,A -85,B 0,C 180,E1 26355.214,E2 26355.214} C_VEL
LIN {X 0,Y 560.212,Z 433.011,A -85,B 0,C 180,E1 26352.23,E2 26352.23} C_VEL
LIN {X 0,Y 560.214,Z 433.011,A -85,B 0,C 180,E1 26348.867,E2 26348.867} C_VEL
LIN {X 0,Y 560.225,Z 433.002,A -85,B 0,C 180,E1 26345.876,E2 26345.876} C_VEL
LIN {X 0,Y 560.2,Z 433.011,A -85,B 0,C 180,E1 26342.581,E2 26342.581} C_VEL
LIN {X 0,Y 560.247,Z 433.012,A -85,B 0,C 180,E1 26339.542,E2 26339.542} C_VEL
LIN {X 0,Y 560.196,Z 433.011,A -85,B 0,C 180,E1 26336.406,E2 26336.406} C_VEL
LIN {X 0,Y 560.273,Z 433.007,A -85,B 0,C 180,E1 26333.253,E2 26333.253} C_VEL
LIN {X 0,Y 560.2,Z 433.011,A -85,B 0,C 180,E1 26330.128,E2 26330.128} C_VEL
LIN {X 0,Y 560.271,Z 433.008,A -85,B 0,C 180,E1 26327.022,E2 26327.022} C_VEL
LIN {X 0,Y 560.207,Z 433.01,A -85,B 0,C 180,E1 26323.858,E2 26323.858} C_VEL
LIN {X 0,Y 560.246,Z 433.007,A -85,B 0,C 180,E1 26320.648,E2 26320.648} C_VEL
LIN {X 0,Y 560.218,Z 433.01,A -85,B 0,C 180,E1 26317.586,E2 26317.586} C_VEL
LIN {X 0,Y 560.221,Z 433.002,A -85,B 0,C 180,E1 26314.208,E2 26314.208} C_VEL
LIN {X 0,Y 560.249,Z 433.009,A -85,B 0,C 180,E1 26311.169,E2 26311.169} C_VEL
LIN {X 0,Y 560.217,Z 433.005,A -85,B 0,C 180,E1 26307.88,E2 26307.88} C_VEL
LIN {X 0,Y 560.281,Z 433.007,A -85,B 0,C 180,E1 26304.683,E2 26304.683} C_VEL
LIN {X 0,Y 560.223,Z 433.009,A -85,B 0,C 180,E1 26301.462,E2 26301.462} C_VEL
LIN {X 0,Y 560.255,Z 432.997,A -85,B 0,C 180,E1 26298.199,E2 26298.199} C_VEL
LIN {X 0,Y 560.24,Z 433.007,A -85,B 0,C 180,E1 26295.088,E2 26295.088} C_VEL
LIN {X 0,Y 560.234,Z 433.005,A -85,B 0,C 180,E1 26291.739,E2 26291.739} C_VEL
LIN {X 0,Y 560.282,Z 433.002,A -85,B 0,C 180,E1 26288.518,E2 26288.518} C_VEL
LIN {X 0,Y 560.23,Z 433.006,A -85,B 0,C 180,E1 26285.325,E2 26285.325} C_VEL
LIN {X 0,Y 560.276,Z 433,A -85,B 0,C 180,E1 26282.033,E2 26282.033} C_VEL
LIN {X 0,Y 560.251,Z 433.003,A -85,B 0,C 180,E1 26278.773,E2 26278.773} C_VEL
LIN {X 0,Y 560.241,Z 433.006,A -85,B 0,C 180,E1 26275.394,E2 26275.394} C_VEL
LIN {X 0,Y 560.281,Z 433.002,A -85,B 0,C 180,E1 26272.205,E2 26272.205} C_VEL
LIN {X 0,Y 560.239,Z 433.007,A -85,B 0,C 180,E1 26268.989,E2 26268.989} C_VEL
LIN {X 0,Y 560.277,Z 432.997,A -85,B 0,C 180,E1 26265.638,E2 26265.638} C_VEL
LIN {X 0,Y 560.27,Z 433.009,A -85,B 0,C 180,E1 26262.339,E2 26262.339} C_VEL
LIN {X 0,Y 560.247,Z 433.002,A -85,B 0,C 180,E1 26258.969,E2 26258.969} C_VEL
LIN {X 0,Y 560.279,Z 433.005,A -85,B 0,C 180,E1 26255.767,E2 26255.767} C_VEL
LIN {X 0,Y 560.254,Z 433.004,A -85,B 0,C 180,E1 26252.469,E2 26252.469} C_VEL
LIN {X 0,Y 560.265,Z 433.001,A -85,B 0,C 180,E1 26249.071,E2 26249.071} C_VEL
LIN {X 0,Y 560.276,Z 433.006,A -85,B 0,C 180,E1 26245.717,E2 26245.717} C_VEL
LIN {X 0,Y 560.257,Z 433.007,A -85,B 0,C 180,E1 26242.385,E2 26242.385} C_VEL
LIN {X 0,Y 560.278,Z 433.002,A -85,B 0,C 180,E1 26239.015,E2 26239.015} C_VEL
LIN {X 0,Y 560.274,Z 433.007,A -85,B 0,C 180,E1 26235.609,E2 26235.609} C_VEL
LIN {X 0,Y 560.26,Z 433.008,A -85,B 0,C 180,E1 26232.284,E2 26232.284} C_VEL
LIN {X 0,Y 560.279,Z 433.003,A -85,B 0,C 180,E1 26228.915,E2 26228.915} C_VEL
LIN {X 0,Y 560.276,Z 433.011,A -85,B 0,C 180,E1 26225.534,E2 26225.534} C_VEL
LIN {X 0,Y 560.263,Z 433.006,A -85,B 0,C 180,E1 26222.23,E2 26222.23} C_VEL
LIN {X 0,Y 560.342,Z 433.496,A -85,B 0,C 180,E1 26222.018,E2 26222.018} C_VEL
LIN {X 0,Y 564.231,Z 444.746,A -85,B 0,C 180,E1 26220.924,E2 26220.924} C_VEL
LIN {X 0,Y 563.585,Z 488.233,A -85,B 0,C 180,E1 26217.813,E2 26217.813} C_VEL
LIN {X 0,Y 562.775,Z 533.916,A -85,B 0,C 180,E1 26214.566,E2 26214.566} C_VEL
LIN {X 0,Y 562.811,Z 539.309,A -85,B 0,C 180,E1 26214.223,E2 26214.223} C_VEL
LIN {X 0,Y 563.719,Z 546.949,A -85,B 0,C 180,E1 26214.074,E2 26214.074} C_VEL
LIN {X 0,Y 562.89,Z 748.309,A -85,B 0,C 180,E1 26211.355,E2 26211.355} C_VEL
LIN {X 0,Y 562.64,Z 767.332,A -85,B 0,C 180,E1 26210.905,E2 26210.905} C_VEL
LIN {X 0,Y 562.355,Z 785.395,A -85,B 0,C 180,E1 26210.286,E2 26210.286} C_VEL
LIN {X 0,Y 562.021,Z 803.142,A -85,B 0,C 180,E1 26209.48,E2 26209.48} C_VEL
LIN {X 0,Y 561.666,Z 819.771,A -85,B 0,C 180,E1 26208.528,E2 26208.528} C_VEL
LIN {X 0,Y 561.31,Z 835.626,A -85,B 0,C 180,E1 26207.413,E2 26207.413} C_VEL
LIN {X 0,Y 560.955,Z 850.905,A -85,B 0,C 180,E1 26206.111,E2 26206.111} C_VEL
LIN {X 0,Y 560.643,Z 864.944,A -85,B 0,C 180,E1 26204.67,E2 26204.67} C_VEL
LIN {X 0,Y 560.378,Z 878.088,A -85,B 0,C 180,E1 26203.042,E2 26203.042} C_VEL
LIN {X 0,Y 560.188,Z 888.865,A -85,B 0,C 180,E1 26201.427,E2 26201.427} C_VEL
LIN {X 0,Y 560.056,Z 898.508,A -85,B 0,C 180,E1 26199.661,E2 26199.661} C_VEL
LIN {X 0,Y 559.976,Z 906.177,A -85,B 0,C 180,E1 26197.903,E2 26197.903} C_VEL
LIN {X 0,Y 559.935,Z 912.411,A -85,B 0,C 180,E1 26196.048,E2 26196.048} C_VEL
LIN {X 0,Y 559.92,Z 916.876,A -85,B 0,C 180,E1 26194.199,E2 26194.199} C_VEL
LIN {X 0,Y 559.915,Z 919.791,A -85,B 0,C 180,E1 26192.252,E2 26192.252} C_VEL
LIN {X 0,Y 559.908,Z 920.94,A -85,B 0,C 180,E1 26190.307,E2 26190.307} C_VEL
LIN {X 0,Y 559.914,Z 920.348,A -85,B 0,C 180,E1 26188.363,E2 26188.363} C_VEL
LIN {X 0,Y 559.911,Z 918.004,A -85,B 0,C 180,E1 26186.417,E2 26186.417} C_VEL
LIN {X 0,Y 559.926,Z 914.098,A -85,B 0,C 180,E1 26184.569,E2 26184.569} C_VEL
LIN {X 0,Y 559.957,Z 908.469,A -85,B 0,C 180,E1 26182.717,E2 26182.717} C_VEL
LIN {X 0,Y 560.027,Z 901.427,A -85,B 0,C 180,E1 26180.961,E2 26180.961} C_VEL
LIN {X 0,Y 560.136,Z 892.516,A -85,B 0,C 180,E1 26179.197,E2 26179.197} C_VEL
LIN {X 0,Y 560.308,Z 882.152,A -85,B 0,C 180,E1 26177.531,E2 26177.531} C_VEL
LIN {X 0,Y 560.531,Z 870.351,A -85,B 0,C 180,E1 26175.961,E2 26175.961} C_VEL
LIN {X 0,Y 560.823,Z 856.801,A -85,B 0,C 180,E1 26174.459,E2 26174.459} C_VEL
LIN {X 0,Y 561.16,Z 842.031,A -85,B 0,C 180,E1 26173.099,E2 26173.099} C_VEL
LIN {X 0,Y 561.529,Z 826.233,A -85,B 0,C 180,E1 26171.898,E2 26171.898} C_VEL
LIN {X 0,Y 561.879,Z 809.049,A -85,B 0,C 180,E1 26170.834,E2 26170.834} C_VEL
LIN {X 0,Y 562.245,Z 791.807,A -85,B 0,C 180,E1 26169.981,E2 26169.981} C_VEL
LIN {X 0,Y 562.542,Z 773.638,A -85,B 0,C 180,E1 26169.29,E2 26169.29} C_VEL
LIN {X 0,Y 562.809,Z 755.069,A -85,B 0,C 180,E1 26168.784,E2 26168.784} C_VEL
LIN {X 0,Y 562.977,Z 734.88,A -85,B 0,C 180,E1 26168.441,E2 26168.441} C_VEL
LIN {X 0,Y 563.551,Z 543.982,A -85,B 0,C 180,E1 26165.878,E2 26165.878} C_VEL
LIN {X 0,Y 562.723,Z 538.331,A -85,B 0,C 180,E1 26165.739,E2 26165.739} C_VEL
LIN {X 0,Y 563.496,Z 492.907,A -85,B 0,C 180,E1 26162.522,E2 26162.522} C_VEL
LIN {X 0,Y 564.146,Z 451.252,A -85,B 0,C 180,E1 26159.543,E2 26159.543} C_VEL
LIN {X 0,Y 564.191,Z 444.618,A -85,B 0,C 180,E1 26159.064,E2 26159.064} C_VEL
LIN {X 0,Y 560.309,Z 433.306,A -85,B 0,C 180,E1 26157.954,E2 26157.954} C_VEL
LIN {X 0,Y 560.268,Z 433.008,A -85,B 0,C 180,E1 26156.901,E2 26156.901} C_VEL
LIN {X 0,Y 560.264,Z 433.007,A -85,B 0,C 180,E1 26153.597,E2 26153.597} C_VEL
LIN {X 0,Y 560.278,Z 433.01,A -85,B 0,C 180,E1 26150.278,E2 26150.278} C_VEL
LIN {X 0,Y 560.275,Z 433.001,A -85,B 0,C 180,E1 26146.878,E2 26146.878} C_VEL
LIN {X 0,Y 560.264,Z 433.007,A -85,B 0,C 180,E1 26143.54,E2 26143.54} C_VEL
LIN {X 0,Y 560.273,Z 433.009,A -85,B 0,C 180,E1 26140.199,E2 26140.199} C_VEL
LIN {X 0,Y 560.279,Z 433.001,A -85,B 0,C 180,E1 26136.842,E2 26136.842} C_VEL
LIN {X 0,Y 560.264,Z 433.006,A -85,B 0,C 180,E1 26133.466,E2 26133.466} C_VEL
LIN {X 0,Y 560.269,Z 433.005,A -85,B 0,C 180,E1 26130.216,E2 26130.216} C_VEL
LIN {X 0,Y 560.263,Z 433.004,A -85,B 0,C 180,E1 26126.955,E2 26126.955} C_VEL
LIN {X 0,Y 560.279,Z 433.007,A -85,B 0,C 180,E1 26123.562,E2 26123.562} C_VEL
LIN {X 0,Y 560.272,Z 433.003,A -85,B 0,C 180,E1 26120.167,E2 26120.167} C_VEL
LIN {X 0,Y 560.26,Z 433.005,A -85,B 0,C 180,E1 26116.911,E2 26116.911} C_VEL
LIN {X 0,Y 560.274,Z 433.003,A -85,B 0,C 180,E1 26113.625,E2 26113.625} C_VEL
LIN {X 0,Y 560.28,Z 432.999,A -85,B 0,C 180,E1 26110.176,E2 26110.176} C_VEL
LIN {X 0,Y 560.26,Z 433.007,A -85,B 0,C 180,E1 26106.867,E2 26106.867} C_VEL
LIN {X 0,Y 560.271,Z 433.002,A -85,B 0,C 180,E1 26103.581,E2 26103.581} C_VEL
LIN {X 0,Y 560.269,Z 432.999,A -85,B 0,C 180,E1 26100.204,E2 26100.204} C_VEL
LIN {X 0,Y 560.263,Z 433.007,A -85,B 0,C 180,E1 26096.766,E2 26096.766} C_VEL
LIN {X 0,Y 560.273,Z 433.004,A -85,B 0,C 180,E1 26093.441,E2 26093.441} C_VEL
LIN {X 0,Y 560.26,Z 433.001,A -85,B 0,C 180,E1 26090.135,E2 26090.135} C_VEL
LIN {X 0,Y 560.277,Z 433.006,A -85,B 0,C 180,E1 26086.795,E2 26086.795} C_VEL
LIN {X 0,Y 560.276,Z 433.004,A -85,B 0,C 180,E1 26083.399,E2 26083.399} C_VEL
LIN {X 0,Y 560.256,Z 433.005,A -85,B 0,C 180,E1 26080.07,E2 26080.07} C_VEL
LIN {X 0,Y 560.279,Z 433.01,A -85,B 0,C 180,E1 26076.772,E2 26076.772} C_VEL
LIN {X 0,Y 560.26,Z 433.006,A -85,B 0,C 180,E1 26076.304,E2 26076.304} C_VEL
LIN {X 0,Y 559.25,Z 433.13,A -85,B 0,C 180,E1 26075.516,E2 26075.516} C_VEL
LIN {X 0,Y 552.85,Z 433.935,A -85,B 0,C 180,E1 26073.305,E2 26073.305} C_VEL
LIN {X 0,Y 552.339,Z 433.997,A -85,B 0,C 180,E1 26072.729,E2 26072.729} C_VEL
LIN {X 0,Y 552.342,Z 433.991,A -85,B 0,C 180,E1 26069.3,E2 26069.3} C_VEL
LIN {X 0,Y 552.318,Z 433.997,A -85,B 0,C 180,E1 26065.987,E2 26065.987} C_VEL
LIN {X 0,Y 552.339,Z 433.999,A -85,B 0,C 180,E1 26062.626,E2 26062.626} C_VEL
LIN {X 0,Y 552.338,Z 433.998,A -85,B 0,C 180,E1 26059.194,E2 26059.194} C_VEL
LIN {X 0,Y 552.377,Z 434.272,A -85,B 0,C 180,E1 26058.555,E2 26058.555} C_VEL
LIN {X 0,Y 555.013,Z 444.491,A -85,B 0,C 180,E1 26057.156,E2 26057.156} C_VEL
LIN {X 0,Y 554.229,Z 472.792,A -85,B 0,C 180,E1 26053.811,E2 26053.811} C_VEL
LIN {X 0,Y 553.584,Z 502.187,A -85,B 0,C 180,E1 26050.422,E2 26050.422} C_VEL
LIN {X 0,Y 553.055,Z 531.759,A -85,B 0,C 180,E1 26047.093,E2 26047.093} C_VEL
LIN {X 0,Y 552.705,Z 556.846,A -85,B 0,C 180,E1 26044.362,E2 26044.362} C_VEL
LIN {X 0,Y 553.462,Z 564.721,A -85,B 0,C 180,E1 26044.218,E2 26044.218} C_VEL
LIN {X 0,Y 553.129,Z 668.36,A -85,B 0,C 180,E1 26042.844,E2 26042.844} C_VEL
LIN {X 0,Y 553.034,Z 682.539,A -85,B 0,C 180,E1 26042.477,E2 26042.477} C_VEL
LIN {X 0,Y 552.863,Z 696.93,A -85,B 0,C 180,E1 26041.903,E2 26041.903} C_VEL
LIN {X 0,Y 552.646,Z 710.402,A -85,B 0,C 180,E1 26041.16,E2 26041.16} C_VEL
LIN {X 0,Y 552.443,Z 722.861,A -85,B 0,C 180,E1 26040.259,E2 26040.259} C_VEL
LIN {X 0,Y 552.273,Z 734.765,A -85,B 0,C 180,E1 26039.144,E2 26039.144} C_VEL
LIN {X 0,Y 552.129,Z 744.577,A -85,B 0,C 180,E1 26037.971,E2 26037.971} C_VEL
LIN {X 0,Y 552.027,Z 753.002,A -85,B 0,C 180,E1 26036.692,E2 26036.692} C_VEL
LIN {X 0,Y 551.957,Z 760.423,A -85,B 0,C 180,E1 26035.195,E2 26035.195} C_VEL
LIN {X 0,Y 551.928,Z 765.645,A -85,B 0,C 180,E1 26033.714,E2 26033.714} C_VEL
LIN {X 0,Y 551.919,Z 769.082,A -85,B 0,C 180,E1 26032.22,E2 26032.22} C_VEL
LIN {X 0,Y 551.917,Z 770.854,A -85,B 0,C 180,E1 26030.576,E2 26030.576} C_VEL
LIN {X 0,Y 551.915,Z 770.622,A -85,B 0,C 180,E1 26028.973,E2 26028.973} C_VEL
LIN {X 0,Y 551.919,Z 768.741,A -85,B 0,C 180,E1 26027.501,E2 26027.501} C_VEL
LIN {X 0,Y 551.931,Z 765.024,A -85,B 0,C 180,E1 26025.983,E2 26025.983} C_VEL
LIN {X 0,Y 551.961,Z 759.843,A -85,B 0,C 180,E1 26024.584,E2 26024.584} C_VEL
LIN {X 0,Y 552.028,Z 752.849,A -85,B 0,C 180,E1 26023.192,E2 26023.192} C_VEL
LIN {X 0,Y 552.141,Z 743.606,A -85,B 0,C 180,E1 26021.808,E2 26021.808} C_VEL
LIN {X 0,Y 552.29,Z 733.56,A -85,B 0,C 180,E1 26020.641,E2 26020.641} C_VEL
LIN {X 0,Y 552.475,Z 722.022,A -85,B 0,C 180,E1 26019.584,E2 26019.584} C_VEL
LIN {X 0,Y 552.67,Z 709.449,A -85,B 0,C 180,E1 26018.688,E2 26018.688} C_VEL
LIN {X 0,Y 552.878,Z 695.745,A -85,B 0,C 180,E1 26017.952,E2 26017.952} C_VEL
LIN {X 0,Y 553.049,Z 681.587,A -85,B 0,C 180,E1 26017.404,E2 26017.404} C_VEL
LIN {X 0,Y 553.18,Z 666.329,A -85,B 0,C 180,E1 26017.027,E2 26017.027} C_VEL
LIN {X 0,Y 553.241,Z 560.684,A -85,B 0,C 180,E1 26015.633,E2 26015.633} C_VEL
LIN {X 0,Y 552.746,Z 556.545,A -85,B 0,C 180,E1 26015.527,E2 26015.527} C_VEL
LIN {X 0,Y 553.094,Z 525.984,A -85,B 0,C 180,E1 26012.175,E2 26012.175} C_VEL
LIN {X 0,Y 553.679,Z 496.682,A -85,B 0,C 180,E1 26008.862,E2 26008.862} C_VEL
LIN {X 0,Y 554.272,Z 467.821,A -85,B 0,C 180,E1 26005.551,E2 26005.551} C_VEL
LIN {X 0,Y 554.903,Z 444.077,A -85,B 0,C 180,E1 26002.754,E2 26002.754} C_VEL
LIN {X 0,Y 552.318,Z 434.091,A -85,B 0,C 180,E1 26001.344,E2 26001.344} C_VEL
LIN {X 0,Y 552.281,Z 434.001,A -85,B 0,C 180,E1 25998.301,E2 25998.301} C_VEL
LIN {X 0,Y 552.274,Z 434.001,A -85,B 0,C 180,E1 25994.888,E2 25994.888} C_VEL
LIN {X 0,Y 552.318,Z 433.999,A -85,B 0,C 180,E1 25991.749,E2 25991.749} C_VEL
LIN {X 0,Y 552.262,Z 434,A -85,B 0,C 180,E1 25988.527,E2 25988.527} C_VEL
LIN {X 0,Y 552.326,Z 433.994,A -85,B 0,C 180,E1 25985.335,E2 25985.335} C_VEL
LIN {X 0,Y 552.261,Z 433.999,A -85,B 0,C 180,E1 25982.153,E2 25982.153} C_VEL
LIN {X 0,Y 552.278,Z 433.999,A -85,B 0,C 180,E1 25978.816,E2 25978.816} C_VEL
LIN {X 0,Y 552.272,Z 434,A -85,B 0,C 180,E1 25975.83,E2 25975.83} C_VEL
LIN {X 0,Y 552.266,Z 433.998,A -85,B 0,C 180,E1 25972.466,E2 25972.466} C_VEL
LIN {X 0,Y 552.318,Z 434.001,A -85,B 0,C 180,E1 25969.329,E2 25969.329} C_VEL
LIN {X 0,Y 552.264,Z 433.998,A -85,B 0,C 180,E1 25966.099,E2 25966.099} C_VEL
LIN {X 0,Y 552.325,Z 433.993,A -85,B 0,C 180,E1 25962.848,E2 25962.848} C_VEL
LIN {X 0,Y 552.274,Z 433.997,A -85,B 0,C 180,E1 25959.724,E2 25959.724} C_VEL
LIN {X 0,Y 552.286,Z 433.995,A -85,B 0,C 180,E1 25956.3,E2 25956.3} C_VEL
LIN {X 0,Y 552.314,Z 433.992,A -85,B 0,C 180,E1 25953.142,E2 25953.142} C_VEL
LIN {X 0,Y 552.276,Z 433.998,A -85,B 0,C 180,E1 25949.859,E2 25949.859} C_VEL
LIN {X 0,Y 552.341,Z 433.988,A -85,B 0,C 180,E1 25946.676,E2 25946.676} C_VEL
LIN {X 0,Y 552.283,Z 433.996,A -85,B 0,C 180,E1 25943.472,E2 25943.472} C_VEL
LIN {X 0,Y 552.305,Z 433.993,A -85,B 0,C 180,E1 25940.119,E2 25940.119} C_VEL
LIN {X 0,Y 552.315,Z 433.989,A -85,B 0,C 180,E1 25936.946,E2 25936.946} C_VEL
LIN {X 0,Y 552.288,Z 433.996,A -85,B 0,C 180,E1 25933.613,E2 25933.613} C_VEL
LIN {X 0,Y 552.343,Z 433.988,A -85,B 0,C 180,E1 25930.324,E2 25930.324} C_VEL
LIN {X 0,Y 552.297,Z 433.992,A -85,B 0,C 180,E1 25927.072,E2 25927.072} C_VEL
LIN {X 0,Y 552.302,Z 433.994,A -85,B 0,C 180,E1 25923.633,E2 25923.633} C_VEL
LIN {X 0,Y 552.342,Z 433.989,A -85,B 0,C 180,E1 25920.415,E2 25920.415} C_VEL
LIN {X 0,Y 552.298,Z 433.995,A -85,B 0,C 180,E1 25917.095,E2 25917.095} C_VEL
LIN {X 0,Y 552.333,Z 433.988,A -85,B 0,C 180,E1 25913.765,E2 25913.765} C_VEL
LIN {X 0,Y 552.334,Z 433.994,A -85,B 0,C 180,E1 25910.413,E2 25910.413} C_VEL
LIN {X 0,Y 552.304,Z 433.994,A -85,B 0,C 180,E1 25907.134,E2 25907.134} C_VEL
LIN {X 0,Y 552.342,Z 433.991,A -85,B 0,C 180,E1 25903.813,E2 25903.813} C_VEL
LIN {X 0,Y 552.325,Z 433.999,A -85,B 0,C 180,E1 25900.434,E2 25900.434} C_VEL
LIN {X 0,Y 552.314,Z 433.992,A -85,B 0,C 180,E1 25897.094,E2 25897.094} C_VEL
LIN {X 0,Y 552.338,Z 433.99,A -85,B 0,C 180,E1 25893.788,E2 25893.788} C_VEL
LIN {X 0,Y 552.316,Z 433.997,A -85,B 0,C 180,E1 25890.502,E2 25890.502} C_VEL
LIN {X 0,Y 552.331,Z 433.991,A -85,B 0,C 180,E1 25887.107,E2 25887.107} C_VEL
LIN {X 0,Y 552.337,Z 433.996,A -85,B 0,C 180,E1 25883.705,E2 25883.705} C_VEL
LIN {X 0,Y 552.317,Z 433.994,A -85,B 0,C 180,E1 25880.415,E2 25880.415} C_VEL
LIN {X 0,Y 552.339,Z 433.991,A -85,B 0,C 180,E1 25877.106,E2 25877.106} C_VEL
LIN {X 0,Y 552.341,Z 434,A -85,B 0,C 180,E1 25873.75,E2 25873.75} C_VEL
LIN {X 0,Y 552.322,Z 433.996,A -85,B 0,C 180,E1 25870.348,E2 25870.348} C_VEL
LIN {X 0,Y 552.336,Z 433.994,A -85,B 0,C 180,E1 25867.031,E2 25867.031} C_VEL
LIN {X 0,Y 552.337,Z 433.998,A -85,B 0,C 180,E1 25863.622,E2 25863.622} C_VEL
LIN {X 0,Y 552.366,Z 434.241,A -85,B 0,C 180,E1 25862.46,E2 25862.46} C_VEL
LIN {X 0,Y 556.868,Z 448.107,A -85,B 0,C 180,E1 25861.079,E2 25861.079} C_VEL
LIN {X 0,Y 556.114,Z 492.666,A -85,B 0,C 180,E1 25857.87,E2 25857.87} C_VEL
LIN {X 0,Y 555.274,Z 536.279,A -85,B 0,C 180,E1 25854.75,E2 25854.75} C_VEL
LIN {X 0,Y 555.38,Z 539.627,A -85,B 0,C 180,E1 25854.562,E2 25854.562} C_VEL
LIN {X 0,Y 556.41,Z 547.924,A -85,B 0,C 180,E1 25854.397,E2 25854.397} C_VEL
LIN {X 0,Y 555.437,Z 748.309,A -85,B 0,C 180,E1 25851.656,E2 25851.656} C_VEL
LIN {X 0,Y 555.15,Z 767.315,A -85,B 0,C 180,E1 25851.201,E2 25851.201} C_VEL
LIN {X 0,Y 554.811,Z 785.393,A -85,B 0,C 180,E1 25850.575,E2 25850.575} C_VEL
LIN {X 0,Y 554.424,Z 803.038,A -85,B 0,C 180,E1 25849.764,E2 25849.764} C_VEL
LIN {X 0,Y 553.993,Z 819.766,A -85,B 0,C 180,E1 25848.794,E2 25848.794} C_VEL
LIN {X 0,Y 553.575,Z 835.624,A -85,B 0,C 180,E1 25847.665,E2 25847.665} C_VEL
LIN {X 0,Y 553.164,Z 850.554,A -85,B 0,C 180,E1 25846.378,E2 25846.378} C_VEL
LIN {X 0,Y 552.811,Z 864.018,A -85,B 0,C 180,E1 25844.99,E2 25844.99} C_VEL
LIN {X 0,Y 552.497,Z 876.913,A -85,B 0,C 180,E1 25843.394,E2 25843.394} C_VEL
LIN {X 0,Y 552.263,Z 888.229,A -85,B 0,C 180,E1 25841.699,E2 25841.699} C_VEL
LIN {X 0,Y 552.095,Z 898.173,A -85,B 0,C 180,E1 25839.87,E2 25839.87} C_VEL
LIN {X 0,Y 551.991,Z 906.177,A -85,B 0,C 180,E1 25838.018,E2 25838.018} C_VEL
LIN {X 0,Y 551.94,Z 912.412,A -85,B 0,C 180,E1 25836.136,E2 25836.136} C_VEL
LIN {X 0,Y 551.92,Z 916.877,A -85,B 0,C 180,E1 25834.26,E2 25834.26} C_VEL
LIN {X 0,Y 551.915,Z 919.792,A -85,B 0,C 180,E1 25832.284,E2 25832.284} C_VEL
LIN {X 0,Y 551.908,Z 920.94,A -85,B 0,C 180,E1 25830.312,E2 25830.312} C_VEL
LIN {X 0,Y 551.914,Z 920.347,A -85,B 0,C 180,E1 25828.339,E2 25828.339} C_VEL
LIN {X 0,Y 551.912,Z 918.003,A -85,B 0,C 180,E1 25826.365,E2 25826.365} C_VEL
LIN {X 0,Y 551.928,Z 914.098,A -85,B 0,C 180,E1 25824.491,E2 25824.491} C_VEL
LIN {X 0,Y 551.967,Z 908.469,A -85,B 0,C 180,E1 25822.611,E2 25822.611} C_VEL
LIN {X 0,Y 552.054,Z 901.214,A -85,B 0,C 180,E1 25820.781,E2 25820.781} C_VEL
LIN {X 0,Y 552.184,Z 892.517,A -85,B 0,C 180,E1 25819.04,E2 25819.04} C_VEL
LIN {X 0,Y 552.393,Z 881.971,A -85,B 0,C 180,E1 25817.321,E2 25817.321} C_VEL
LIN {X 0,Y 552.654,Z 870.351,A -85,B 0,C 180,E1 25815.756,E2 25815.756} C_VEL
LIN {X 0,Y 553.007,Z 856.576,A -85,B 0,C 180,E1 25814.21,E2 25814.21} C_VEL
LIN {X 0,Y 553.415,Z 841.604,A -85,B 0,C 180,E1 25812.819,E2 25812.819} C_VEL
LIN {X 0,Y 553.853,Z 825.435,A -85,B 0,C 180,E1 25811.584,E2 25811.584} C_VEL
LIN {X 0,Y 554.256,Z 809.051,A -85,B 0,C 180,E1 25810.559,E2 25810.559} C_VEL
LIN {X 0,Y 554.678,Z 791.809,A -85,B 0,C 180,E1 25809.696,E2 25809.696} C_VEL
LIN {X 0,Y 555.034,Z 773.533,A -85,B 0,C 180,E1 25808.993,E2 25808.993} C_VEL
LIN {X 0,Y 555.344,Z 754.923,A -85,B 0,C 180,E1 25808.482,E2 25808.482} C_VEL
LIN {X 0,Y 555.54,Z 734.498,A -85,B 0,C 180,E1 25808.132,E2 25808.132} C_VEL
LIN {X 0,Y 556.238,Z 545.044,A -85,B 0,C 180,E1 25805.555,E2 25805.555} C_VEL
LIN {X 0,Y 555.251,Z 538.376,A -85,B 0,C 180,E1 25805.394,E2 25805.394} C_VEL
LIN {X 0,Y 556.098,Z 493.703,A -85,B 0,C 180,E1 25802.204,E2 25802.204} C_VEL
LIN {X 0,Y 556.844,Z 448.887,A -85,B 0,C 180,E1 25798.981,E2 25798.981} C_VEL
LIN {X 0,Y 556.53,Z 446.513,A -85,B 0,C 180,E1 25798.779,E2 25798.779} C_VEL
LIN {X 0,Y 552.364,Z 434.226,A -85,B 0,C 180,E1 25797.54,E2 25797.54} C_VEL
LIN {X 0,Y 552.34,Z 433.999,A -85,B 0,C 180,E1 25794.218,E2 25794.218} C_VEL
LIN {X 0,Y 552.33,Z 433.993,A -85,B 0,C 180,E1 25790.786,E2 25790.786} C_VEL
LIN {X 0,Y 552.325,Z 433.992,A -85,B 0,C 180,E1 25787.458,E2 25787.458} C_VEL
LIN {X 0,Y 552.341,Z 433.998,A -85,B 0,C 180,E1 25784.037,E2 25784.037} C_VEL
LIN {X 0,Y 552.334,Z 433.993,A -85,B 0,C 180,E1 25780.669,E2 25780.669} C_VEL
LIN {X 0,Y 552.324,Z 433.995,A -85,B 0,C 180,E1 25777.333,E2 25777.333} C_VEL
LIN {X 0,Y 552.337,Z 433.998,A -85,B 0,C 180,E1 25773.995,E2 25773.995} C_VEL
LIN {X 0,Y 552.339,Z 433.991,A -85,B 0,C 180,E1 25770.575,E2 25770.575} C_VEL
LIN {X 0,Y 552.324,Z 433.995,A -85,B 0,C 180,E1 25767.258,E2 25767.258} C_VEL
LIN {X 0,Y 552.334,Z 433.994,A -85,B 0,C 180,E1 25763.912,E2 25763.912} C_VEL
LIN {X 0,Y 552.338,Z 433.989,A -85,B 0,C 180,E1 25760.56,E2 25760.56} C_VEL
LIN {X 0,Y 552.325,Z 433.997,A -85,B 0,C 180,E1 25757.162,E2 25757.162} C_VEL
LIN {X 0,Y 552.331,Z 433.989,A -85,B 0,C 180,E1 25753.825,E2 25753.825} C_VEL
LIN {X 0,Y 552.325,Z 433.989,A -85,B 0,C 180,E1 25750.535,E2 25750.535} C_VEL
LIN {X 0,Y 552.33,Z 433.998,A -85,B 0,C 180,E1 25747.071,E2 25747.071} C_VEL
LIN {X 0,Y 552.333,Z 433.989,A -85,B 0,C 180,E1 25743.736,E2 25743.736} C_VEL
LIN {X 0,Y 552.321,Z 433.989,A -85,B 0,C 180,E1 25740.415,E2 25740.415} C_VEL
LIN {X 0,Y 552.335,Z 433.998,A -85,B 0,C 180,E1 25736.991,E2 25736.991} C_VEL
LIN {X 0,Y 552.335,Z 433.991,A -85,B 0,C 180,E1 25733.556,E2 25733.556} C_VEL
LIN {X 0,Y 552.318,Z 433.991,A -85,B 0,C 180,E1 25730.307,E2 25730.307} C_VEL
LIN {X 0,Y 552.34,Z 433.996,A -85,B 0,C 180,E1 25726.922,E2 25726.922} C_VEL
LIN {X 0,Y 552.34,Z 433.992,A -85,B 0,C 180,E1 25723.488,E2 25723.488} C_VEL
LIN {X 0,Y 552.317,Z 433.994,A -85,B 0,C 180,E1 25720.102,E2 25720.102} C_VEL
LIN {X 0,Y 552.341,Z 434,A -85,B 0,C 180,E1 25716.757,E2 25716.757} C_VEL
LIN {X 0,Y 552.341,Z 433.992,A -85,B 0,C 180,E1 25713.324,E2 25713.324} C_VEL
LIN {X 0,Y 552.339,Z 433.997,A -85,B 0,C 180,E1 25712.729,E2 25712.729} C_VEL
LIN {X 0,Y 551.375,Z 434.116,A -85,B 0,C 180,E1 25711.93,E2 25711.93} C_VEL
LIN {X 0,Y 544.85,Z 434.925,A -85,B 0,C 180,E1 25709.628,E2 25709.628} C_VEL
LIN {X 0,Y 544.4,Z 434.982,A -85,B 0,C 180,E1 25709.102,E2 25709.102} C_VEL
LIN {X 0,Y 544.378,Z 434.984,A -85,B 0,C 180,E1 25705.742,E2 25705.742} C_VEL
LIN {X 0,Y 544.399,Z 434.986,A -85,B 0,C 180,E1 25702.294,E2 25702.294} C_VEL
LIN {X 0,Y 544.435,Z 435.214,A -85,B 0,C 180,E1 25698.942,E2 25698.942} C_VEL
